LIN {X 0,Y 369.311,Z 529.296,A -85,B 0,C 180,E1 -12777.819,E2 -12777.819} C_VEL
LIN {X 0,Y 369.451,Z 529.279,A -85,B 0,C 180,E1 -12780,E2 -12780} C_VEL
LIN {X 0,Y 369.322,Z 529.581,A -85,B 0,C 180,E1 -12780.716,E2 -12780.716} C_VEL
LIN {X 0,Y 369.615,Z 530.776,A -85,B 0,C 180,E1 -12780.886,E2 -12780.886} C_VEL
LIN {X 0,Y 374.788,Z 542.535,A -85,B 0,C 180,E1 -12781.531,E2 -12781.531} C_VEL
LIN {X 0,Y 376.428,Z 547.392,A -85,B 0,C 180,E1 -12781.75,E2 -12781.75} C_VEL
LIN {X 0,Y 376.481,Z 569.423,A -85,B 0,C 180,E1 -12782.286,E2 -12782.286} C_VEL
LIN {X 0,Y 376.386,Z 581.867,A -85,B 0,C 180,E1 -12782.806,E2 -12782.806} C_VEL
LIN {X 0,Y 376.073,Z 593.193,A -85,B 0,C 180,E1 -12783.482,E2 -12783.482} C_VEL
LIN {X 0,Y 375.404,Z 605.188,A -85,B 0,C 180,E1 -12784.429,E2 -12784.429} C_VEL
LIN {X 0,Y 374.736,Z 615.62,A -85,B 0,C 180,E1 -12785.499,E2 -12785.499} C_VEL
LIN {X 0,Y 373.913,Z 625.309,A -85,B 0,C 180,E1 -12786.747,E2 -12786.747} C_VEL
LIN {X 0,Y 373.096,Z 633.924,A -85,B 0,C 180,E1 -12788.122,E2 -12788.122} C_VEL
LIN {X 0,Y 372.293,Z 640.997,A -85,B 0,C 180,E1 -12789.508,E2 -12789.508} C_VEL
LIN {X 0,Y 371.594,Z 646.791,A -85,B 0,C 180,E1 -12790.903,E2 -12790.903} C_VEL
LIN {X 0,Y 370.872,Z 652.348,A -85,B 0,C 180,E1 -12792.588,E2 -12792.588} C_VEL
LIN {X 0,Y 370.18,Z 657.037,A -85,B 0,C 180,E1 -12794.481,E2 -12794.481} C_VEL
LIN {X 0,Y 369.897,Z 658.839,A -85,B 0,C 180,E1 -12795.427,E2 -12795.427} C_VEL
LIN {X 0,Y 369.624,Z 660.529,A -85,B 0,C 180,E1 -12796.572,E2 -12796.572} C_VEL
LIN {X 0,Y 369.348,Z 661.936,A -85,B 0,C 180,E1 -12797.94,E2 -12797.94} C_VEL
LIN {X 0,Y 369.231,Z 662.502,A -85,B 0,C 180,E1 -12798.88,E2 -12798.88} C_VEL
LIN {X 0,Y 369.092,Z 662.755,A -85,B 0,C 180,E1 -12800.045,E2 -12800.045} C_VEL
LIN {X 0,Y 369.016,Z 662.563,A -85,B 0,C 180,E1 -12801.215,E2 -12801.215} C_VEL
LIN {X 0,Y 368.966,Z 661.866,A -85,B 0,C 180,E1 -12802.393,E2 -12802.393} C_VEL
LIN {X 0,Y 369.024,Z 660.255,A -85,B 0,C 180,E1 -12803.918,E2 -12803.918} C_VEL
LIN {X 0,Y 369.263,Z 656.737,A -85,B 0,C 180,E1 -12805.961,E2 -12805.961} C_VEL
LIN {X 0,Y 369.574,Z 652.281,A -85,B 0,C 180,E1 -12807.769,E2 -12807.769} C_VEL
LIN {X 0,Y 370.008,Z 646.26,A -85,B 0,C 180,E1 -12809.594,E2 -12809.594} C_VEL
LIN {X 0,Y 370.55,Z 638.583,A -85,B 0,C 180,E1 -12811.409,E2 -12811.409} C_VEL
LIN {X 0,Y 371.201,Z 630.13,A -85,B 0,C 180,E1 -12812.979,E2 -12812.979} C_VEL
LIN {X 0,Y 371.811,Z 620.701,A -85,B 0,C 180,E1 -12814.4,E2 -12814.4} C_VEL
LIN {X 0,Y 372.43,Z 610.239,A -85,B 0,C 180,E1 -12815.664,E2 -12815.664} C_VEL
LIN {X 0,Y 373.009,Z 599.015,A -85,B 0,C 180,E1 -12816.743,E2 -12816.743} C_VEL
LIN {X 0,Y 373.444,Z 588.322,A -85,B 0,C 180,E1 -12817.554,E2 -12817.554} C_VEL
LIN {X 0,Y 373.76,Z 575.886,A -85,B 0,C 180,E1 -12818.266,E2 -12818.266} C_VEL
LIN {X 0,Y 373.907,Z 562.29,A -85,B 0,C 180,E1 -12818.796,E2 -12818.796} C_VEL
LIN {X 0,Y 373.805,Z 544.593,A -85,B 0,C 180,E1 -12819.216,E2 -12819.216} C_VEL
LIN {X 0,Y 369.179,Z 530.472,A -85,B 0,C 180,E1 -12819.719,E2 -12819.719} C_VEL
LIN {X 0,Y 368.967,Z 529.473,A -85,B 0,C 180,E1 -12819.913,E2 -12819.913} C_VEL
LIN {X 0,Y 368.887,Z 529.349,A -85,B 0,C 180,E1 -12823.618,E2 -12823.618} C_VEL
LIN {X 0,Y 368.937,Z 529.338,A -85,B 0,C 180,E1 -12826.705,E2 -12826.705} C_VEL
LIN {X 0,Y 368.952,Z 529.339,A -85,B 0,C 180,E1 -12829.637,E2 -12829.637} C_VEL
LIN {X 0,Y 368.903,Z 529.345,A -85,B 0,C 180,E1 -12833.145,E2 -12833.145} C_VEL
LIN {X 0,Y 368.897,Z 529.342,A -85,B 0,C 180,E1 -12836.463,E2 -12836.463} C_VEL
LIN {X 0,Y 368.93,Z 529.34,A -85,B 0,C 180,E1 -12839.047,E2 -12839.047} C_VEL
LIN {X 0,Y 368.981,Z 529.338,A -85,B 0,C 180,E1 -12841.565,E2 -12841.565} C_VEL
LIN {X 0,Y 369.002,Z 529.331,A -85,B 0,C 180,E1 -12844.021,E2 -12844.021} C_VEL
LIN {X 0,Y 368.936,Z 529.344,A -85,B 0,C 180,E1 -12847.606,E2 -12847.606} C_VEL
LIN {X 0,Y 368.958,Z 529.336,A -85,B 0,C 180,E1 -12851.106,E2 -12851.106} C_VEL
LIN {X 0,Y 369.001,Z 529.329,A -85,B 0,C 180,E1 -12854.536,E2 -12854.536} C_VEL
LIN {X 0,Y 369.009,Z 529.332,A -85,B 0,C 180,E1 -12857.907,E2 -12857.907} C_VEL
LIN {X 0,Y 369.098,Z 529.319,A -85,B 0,C 180,E1 -12861.238,E2 -12861.238} C_VEL
LIN {X 0,Y 369.135,Z 529.313,A -85,B 0,C 180,E1 -12864.538,E2 -12864.538} C_VEL
LIN {X 0,Y 369.321,Z 529.295,A -85,B 0,C 180,E1 -12867.819,E2 -12867.819} C_VEL
LIN {X 0,Y 369.461,Z 529.276,A -85,B 0,C 180,E1 -12870,E2 -12870} C_VEL
LIN {X 0,Y 369.321,Z 529.292,A -85,B 0,C 180,E1 -12872.181,E2 -12872.181} C_VEL
LIN {X 0,Y 369.178,Z 529.308,A -85,B 0,C 180,E1 -12876.559,E2 -12876.559} C_VEL
LIN {X 0,Y 369.068,Z 529.327,A -85,B 0,C 180,E1 -12879.868,E2 -12879.868} C_VEL
LIN {X 0,Y 369.041,Z 529.33,A -85,B 0,C 180,E1 -12883.772,E2 -12883.772} C_VEL
LIN {X 0,Y 369.005,Z 529.334,A -85,B 0,C 180,E1 -12887.768,E2 -12887.768} C_VEL
LIN {X 0,Y 368.9,Z 529.341,A -85,B 0,C 180,E1 -12891.574,E2 -12891.574} C_VEL
LIN {X 0,Y 368.957,Z 529.335,A -85,B 0,C 180,E1 -12894.775,E2 -12894.775} C_VEL
LIN {X 0,Y 368.986,Z 529.334,A -85,B 0,C 180,E1 -12896.321,E2 -12896.321} C_VEL
LIN {X 0,Y 368.299,Z 529.418,A -85,B 0,C 180,E1 -12897.231,E2 -12897.231} C_VEL
LIN {X 0,Y 365.402,Z 529.778,A -85,B 0,C 180,E1 -12898.711,E2 -12898.711} C_VEL
LIN {X 0,Y 362.962,Z 530.087,A -85,B 0,C 180,E1 -12899.908,E2 -12899.908} C_VEL
LIN {X 0,Y 361.925,Z 530.211,A -85,B 0,C 180,E1 -12900.834,E2 -12900.834} C_VEL
LIN {X 0,Y 361.846,Z 530.221,A -85,B 0,C 180,E1 -12901.148,E2 -12901.148} C_VEL
LIN {X 0,Y 361.856,Z 530.223,A -85,B 0,C 180,E1 -12904.279,E2 -12904.279} C_VEL
LIN {X 0,Y 361.866,Z 530.218,A -85,B 0,C 180,E1 -12907.222,E2 -12907.222} C_VEL
LIN {X 0,Y 361.906,Z 530.214,A -85,B 0,C 180,E1 -12910.767,E2 -12910.767} C_VEL
LIN {X 0,Y 361.91,Z 530.216,A -85,B 0,C 180,E1 -12914.353,E2 -12914.353} C_VEL
LIN {X 0,Y 361.835,Z 530.223,A -85,B 0,C 180,E1 -12917.567,E2 -12917.567} C_VEL
LIN {X 0,Y 361.868,Z 530.218,A -85,B 0,C 180,E1 -12920.972,E2 -12920.972} C_VEL
LIN {X 0,Y 361.871,Z 530.219,A -85,B 0,C 180,E1 -12924.654,E2 -12924.654} C_VEL
LIN {X 0,Y 361.857,Z 530.224,A -85,B 0,C 180,E1 -12928.372,E2 -12928.372} C_VEL
LIN {X 0,Y 361.919,Z 530.218,A -85,B 0,C 180,E1 -12932.221,E2 -12932.221} C_VEL
LIN {X 0,Y 361.923,Z 530.213,A -85,B 0,C 180,E1 -12934.709,E2 -12934.709} C_VEL
LIN {X 0,Y 361.894,Z 530.221,A -85,B 0,C 180,E1 -12938.347,E2 -12938.347} C_VEL
LIN {X 0,Y 361.962,Z 530.21,A -85,B 0,C 180,E1 -12942.06,E2 -12942.06} C_VEL
LIN {X 0,Y 361.992,Z 530.206,A -85,B 0,C 180,E1 -12946.1,E2 -12946.1} C_VEL
LIN {X 0,Y 362.029,Z 530.2,A -85,B 0,C 180,E1 -12949.937,E2 -12949.937} C_VEL
LIN {X 0,Y 362.145,Z 530.187,A -85,B 0,C 180,E1 -12952.192,E2 -12952.192} C_VEL
LIN {X 0,Y 362.113,Z 530.194,A -85,B 0,C 180,E1 -12954.431,E2 -12954.431} C_VEL
LIN {X 0,Y 362.276,Z 530.168,A -85,B 0,C 180,E1 -12957.776,E2 -12957.776} C_VEL
LIN {X 0,Y 362.42,Z 530.151,A -85,B 0,C 180,E1 -12960,E2 -12960} C_VEL
LIN {X 0,Y 362.275,Z 530.171,A -85,B 0,C 180,E1 -12962.223,E2 -12962.223} C_VEL
LIN {X 0,Y 362.155,Z 530.187,A -85,B 0,C 180,E1 -12966.686,E2 -12966.686} C_VEL
LIN {X 0,Y 362.023,Z 530.2,A -85,B 0,C 180,E1 -12970.062,E2 -12970.062} C_VEL
LIN {X 0,Y 361.99,Z 530.203,A -85,B 0,C 180,E1 -12973.899,E2 -12973.899} C_VEL
LIN {X 0,Y 361.96,Z 530.207,A -85,B 0,C 180,E1 -12977.939,E2 -12977.939} C_VEL
LIN {X 0,Y 361.854,Z 530.219,A -85,B 0,C 180,E1 -12981.655,E2 -12981.655} C_VEL
LIN {X 0,Y 361.92,Z 530.212,A -85,B 0,C 180,E1 -12985.29,E2 -12985.29} C_VEL
LIN {X 0,Y 361.916,Z 530.212,A -85,B 0,C 180,E1 -12987.778,E2 -12987.778} C_VEL
LIN {X 0,Y 361.84,Z 530.223,A -85,B 0,C 180,E1 -12991.285,E2 -12991.285} C_VEL
LIN {X 0,Y 361.848,Z 530.222,A -85,B 0,C 180,E1 -12994.281,E2 -12994.281} C_VEL
LIN {X 0,Y 361.859,Z 530.221,A -85,B 0,C 180,E1 -12997.223,E2 -12997.223} C_VEL
LIN {X 0,Y 361.83,Z 530.228,A -85,B 0,C 180,E1 -13000.756,E2 -13000.756} C_VEL
LIN {X 0,Y 361.83,Z 530.224,A -85,B 0,C 180,E1 -13004.366,E2 -13004.366} C_VEL
LIN {X 0,Y 361.832,Z 530.223,A -85,B 0,C 180,E1 -13007.568,E2 -13007.568} C_VEL
LIN {X 0,Y 361.868,Z 530.224,A -85,B 0,C 180,E1 -13010.973,E2 -13010.973} C_VEL
LIN {X 0,Y 361.875,Z 530.224,A -85,B 0,C 180,E1 -13014.655,E2 -13014.655} C_VEL
LIN {X 0,Y 361.97,Z 530.418,A -85,B 0,C 180,E1 -13015.791,E2 -13015.791} C_VEL
LIN {X 0,Y 364.841,Z 544.913,A -85,B 0,C 180,E1 -13019.626,E2 -13019.626} C_VEL
LIN {X 0,Y 365.525,Z 550.193,A -85,B 0,C 180,E1 -13020.956,E2 -13020.956} C_VEL
LIN {X 0,Y 364.093,Z 565.356,A -85,B 0,C 180,E1 -13024.566,E2 -13024.566} C_VEL
LIN {X 0,Y 362.582,Z 584.16,A -85,B 0,C 180,E1 -13028.987,E2 -13028.987} C_VEL
LIN {X 0,Y 361.692,Z 599.262,A -85,B 0,C 180,E1 -13032.463,E2 -13032.463} C_VEL
LIN {X 0,Y 363.071,Z 616.076,A -85,B 0,C 180,E1 -13032.992,E2 -13032.992} C_VEL
LIN {X 0,Y 365.581,Z 647.576,A -85,B 0,C 180,E1 -13033.892,E2 -13033.892} C_VEL
LIN {X 0,Y 364.865,Z 683.205,A -85,B 0,C 180,E1 -13034.821,E2 -13034.821} C_VEL
LIN {X 0,Y 364.369,Z 695.019,A -85,B 0,C 180,E1 -13035.336,E2 -13035.336} C_VEL
LIN {X 0,Y 363.573,Z 705.872,A -85,B 0,C 180,E1 -13036.018,E2 -13036.018} C_VEL
LIN {X 0,Y 363.02,Z 715.883,A -85,B 0,C 180,E1 -13036.852,E2 -13036.852} C_VEL
LIN {X 0,Y 362.191,Z 726.2,A -85,B 0,C 180,E1 -13037.96,E2 -13037.96} C_VEL
LIN {X 0,Y 361.582,Z 734.455,A -85,B 0,C 180,E1 -13039.076,E2 -13039.076} C_VEL
LIN {X 0,Y 361.212,Z 742.776,A -85,B 0,C 180,E1 -13040.481,E2 -13040.481} C_VEL
LIN {X 0,Y 361.042,Z 749.412,A -85,B 0,C 180,E1 -13041.887,E2 -13041.887} C_VEL
LIN {X 0,Y 361.026,Z 754.682,A -85,B 0,C 180,E1 -13043.293,E2 -13043.293} C_VEL
LIN {X 0,Y 361.121,Z 759.526,A -85,B 0,C 180,E1 -13044.976,E2 -13044.976} C_VEL
LIN {X 0,Y 361.292,Z 762.876,A -85,B 0,C 180,E1 -13046.654,E2 -13046.654} C_VEL
LIN {X 0,Y 361.355,Z 764.387,A -85,B 0,C 180,E1 -13047.771,E2 -13047.771} C_VEL
LIN {X 0,Y 361.435,Z 765.3,A -85,B 0,C 180,E1 -13048.886,E2 -13048.886} C_VEL
LIN {X 0,Y 361.683,Z 765.721,A -85,B 0,C 180,E1 -13050,E2 -13050} C_VEL
LIN {X 0,Y 361.405,Z 765.487,A -85,B 0,C 180,E1 -13051.114,E2 -13051.114} C_VEL
LIN {X 0,Y 361.299,Z 764.759,A -85,B 0,C 180,E1 -13052.229,E2 -13052.229} C_VEL
LIN {X 0,Y 361.247,Z 763.478,A -85,B 0,C 180,E1 -13053.346,E2 -13053.346} C_VEL
LIN {X 0,Y 361.011,Z 760.507,A -85,B 0,C 180,E1 -13055.026,E2 -13055.026} C_VEL
LIN {X 0,Y 360.857,Z 756.183,A -85,B 0,C 180,E1 -13056.71,E2 -13056.71} C_VEL
LIN {X 0,Y 360.96,Z 750.431,A -85,B 0,C 180,E1 -13058.396,E2 -13058.396} C_VEL
LIN {X 0,Y 361.297,Z 742.939,A -85,B 0,C 180,E1 -13060.082,E2 -13060.082} C_VEL
LIN {X 0,Y 361.872,Z 735.075,A -85,B 0,C 180,E1 -13061.482,E2 -13061.482} C_VEL
LIN {X 0,Y 362.806,Z 725.285,A -85,B 0,C 180,E1 -13062.871,E2 -13062.871} C_VEL
LIN {X 0,Y 363.901,Z 714.064,A -85,B 0,C 180,E1 -13064.112,E2 -13064.112} C_VEL
LIN {X 0,Y 364.995,Z 702.831,A -85,B 0,C 180,E1 -13065.066,E2 -13065.066} C_VEL
LIN {X 0,Y 365.976,Z 690.812,A -85,B 0,C 180,E1 -13065.832,E2 -13065.832} C_VEL
LIN {X 0,Y 366.787,Z 678.323,A -85,B 0,C 180,E1 -13066.387,E2 -13066.387} C_VEL
LIN {X 0,Y 367.347,Z 657.774,A -85,B 0,C 180,E1 -13066.933,E2 -13066.933} C_VEL
LIN {X 0,Y 367.41,Z 645.582,A -85,B 0,C 180,E1 -13067.245,E2 -13067.245} C_VEL
LIN {X 0,Y 365.873,Z 619.079,A -85,B 0,C 180,E1 -13068.042,E2 -13068.042} C_VEL
LIN {X 0,Y 363.361,Z 597.729,A -85,B 0,C 180,E1 -13068.795,E2 -13068.795} C_VEL
LIN {X 0,Y 361.865,Z 587.816,A -85,B 0,C 180,E1 -13069.216,E2 -13069.216} C_VEL
LIN {X 0,Y 362.492,Z 575.864,A -85,B 0,C 180,E1 -13071.914,E2 -13071.914} C_VEL
LIN {X 0,Y 363.779,Z 558.36,A -85,B 0,C 180,E1 -13076.072,E2 -13076.072} C_VEL
LIN {X 0,Y 364.81,Z 547.337,A -85,B 0,C 180,E1 -13078.79,E2 -13078.79} C_VEL
LIN {X 0,Y 364.315,Z 542.419,A -85,B 0,C 180,E1 -13080.103,E2 -13080.103} C_VEL
LIN {X 0,Y 362.061,Z 530.888,A -85,B 0,C 180,E1 -13083.418,E2 -13083.418} C_VEL
LIN {X 0,Y 361.927,Z 530.221,A -85,B 0,C 180,E1 -13083.776,E2 -13083.776} C_VEL
LIN {X 0,Y 361.86,Z 530.224,A -85,B 0,C 180,E1 -13087.223,E2 -13087.223} C_VEL
LIN {X 0,Y 361.831,Z 530.226,A -85,B 0,C 180,E1 -13090.755,E2 -13090.755} C_VEL
LIN {X 0,Y 361.842,Z 530.223,A -85,B 0,C 180,E1 -13094.363,E2 -13094.363} C_VEL
LIN {X 0,Y 361.878,Z 530.214,A -85,B 0,C 180,E1 -13097.559,E2 -13097.559} C_VEL
LIN {X 0,Y 361.87,Z 530.217,A -85,B 0,C 180,E1 -13100.971,E2 -13100.971} C_VEL
LIN {X 0,Y 361.868,Z 530.216,A -85,B 0,C 180,E1 -13104.655,E2 -13104.655} C_VEL
LIN {X 0,Y 361.853,Z 530.22,A -85,B 0,C 180,E1 -13108.372,E2 -13108.372} C_VEL
LIN {X 0,Y 361.915,Z 530.215,A -85,B 0,C 180,E1 -13112.222,E2 -13112.222} C_VEL
LIN {X 0,Y 361.92,Z 530.213,A -85,B 0,C 180,E1 -13114.71,E2 -13114.71} C_VEL
LIN {X 0,Y 361.885,Z 530.22,A -85,B 0,C 180,E1 -13118.347,E2 -13118.347} C_VEL
LIN {X 0,Y 361.959,Z 530.207,A -85,B 0,C 180,E1 -13122.061,E2 -13122.061} C_VEL
LIN {X 0,Y 361.99,Z 530.207,A -85,B 0,C 180,E1 -13126.101,E2 -13126.101} C_VEL
LIN {X 0,Y 362.028,Z 530.203,A -85,B 0,C 180,E1 -13129.938,E2 -13129.938} C_VEL
LIN {X 0,Y 362.143,Z 530.19,A -85,B 0,C 180,E1 -13132.193,E2 -13132.193} C_VEL
LIN {X 0,Y 362.116,Z 530.191,A -85,B 0,C 180,E1 -13134.432,E2 -13134.432} C_VEL
LIN {X 0,Y 362.275,Z 530.173,A -85,B 0,C 180,E1 -13137.777,E2 -13137.777} C_VEL
LIN {X 0,Y 362.391,Z 530.263,A -85,B 0,C 180,E1 -13140.125,E2 -13140.125} C_VEL
LIN {X 0,Y 362.532,Z 531.164,A -85,B 0,C 180,E1 -13140.344,E2 -13140.344} C_VEL
LIN {X 0,Y 368.491,Z 544.802,A -85,B 0,C 180,E1 -13141.139,E2 -13141.139} C_VEL
LIN {X 0,Y 369.944,Z 548.817,A -85,B 0,C 180,E1 -13141.334,E2 -13141.334} C_VEL
LIN {X 0,Y 370.011,Z 570.604,A -85,B 0,C 180,E1 -13141.875,E2 -13141.875} C_VEL
LIN {X 0,Y 369.898,Z 583.228,A -85,B 0,C 180,E1 -13142.413,E2 -13142.413} C_VEL
LIN {X 0,Y 369.509,Z 595.258,A -85,B 0,C 180,E1 -13143.157,E2 -13143.157} C_VEL
LIN {X 0,Y 368.803,Z 606.791,A -85,B 0,C 180,E1 -13144.098,E2 -13144.098} C_VEL
LIN {X 0,Y 368.09,Z 617.219,A -85,B 0,C 180,E1 -13145.204,E2 -13145.204} C_VEL
LIN {X 0,Y 367.12,Z 627.66,A -85,B 0,C 180,E1 -13146.596,E2 -13146.596} C_VEL
LIN {X 0,Y 366.269,Z 636.06,A -85,B 0,C 180,E1 -13147.997,E2 -13147.997} C_VEL
LIN {X 0,Y 365.246,Z 644.156,A -85,B 0,C 180,E1 -13149.693,E2 -13149.693} C_VEL
LIN {X 0,Y 364.561,Z 649.571,A -85,B 0,C 180,E1 -13151.115,E2 -13151.115} C_VEL
LIN {X 0,Y 363.801,Z 654.789,A -85,B 0,C 180,E1 -13152.836,E2 -13152.836} C_VEL
LIN {X 0,Y 363.165,Z 658.84,A -85,B 0,C 180,E1 -13154.629,E2 -13154.629} C_VEL
LIN {X 0,Y 362.845,Z 660.682,A -85,B 0,C 180,E1 -13155.734,E2 -13155.734} C_VEL
LIN {X 0,Y 362.552,Z 662.185,A -85,B 0,C 180,E1 -13156.905,E2 -13156.905} C_VEL
LIN {X 0,Y 362.314,Z 663.202,A -85,B 0,C 180,E1 -13158.111,E2 -13158.111} C_VEL
LIN {X 0,Y 362.171,Z 663.712,A -85,B 0,C 180,E1 -13159.262,E2 -13159.262} C_VEL
LIN {X 0,Y 361.999,Z 663.563,A -85,B 0,C 180,E1 -13161.272,E2 -13161.272} C_VEL
LIN {X 0,Y 361.945,Z 662.47,A -85,B 0,C 180,E1 -13162.852,E2 -13162.852} C_VEL
LIN {X 0,Y 362.032,Z 660.894,A -85,B 0,C 180,E1 -13164.165,E2 -13164.165} C_VEL
LIN {X 0,Y 362.221,Z 657.929,A -85,B 0,C 180,E1 -13165.885,E2 -13165.885} C_VEL
LIN {X 0,Y 362.542,Z 653.515,A -85,B 0,C 180,E1 -13167.727,E2 -13167.727} C_VEL
LIN {X 0,Y 363.012,Z 647.024,A -85,B 0,C 180,E1 -13169.731,E2 -13169.731} C_VEL
LIN {X 0,Y 363.555,Z 639.803,A -85,B 0,C 180,E1 -13171.463,E2 -13171.463} C_VEL
LIN {X 0,Y 364.19,Z 631.558,A -85,B 0,C 180,E1 -13173.036,E2 -13173.036} C_VEL
LIN {X 0,Y 364.843,Z 621.635,A -85,B 0,C 180,E1 -13174.563,E2 -13174.563} C_VEL
LIN {X 0,Y 365.488,Z 611.245,A -85,B 0,C 180,E1 -13175.838,E2 -13175.838} C_VEL
LIN {X 0,Y 366.053,Z 600.766,A -85,B 0,C 180,E1 -13176.869,E2 -13176.869} C_VEL
LIN {X 0,Y 366.543,Z 589.314,A -85,B 0,C 180,E1 -13177.761,E2 -13177.761} C_VEL
LIN {X 0,Y 366.86,Z 577.017,A -85,B 0,C 180,E1 -13178.478,E2 -13178.478} C_VEL
LIN {X 0,Y 367.009,Z 563.458,A -85,B 0,C 180,E1 -13179.02,E2 -13179.02} C_VEL
LIN {X 0,Y 366.849,Z 545.757,A -85,B 0,C 180,E1 -13179.453,E2 -13179.453} C_VEL
LIN {X 0,Y 362.055,Z 531.081,A -85,B 0,C 180,E1 -13180.003,E2 -13180.003} C_VEL
LIN {X 0,Y 361.897,Z 530.288,A -85,B 0,C 180,E1 -13180.221,E2 -13180.221} C_VEL
LIN {X 0,Y 361.836,Z 530.225,A -85,B 0,C 180,E1 -13184.058,E2 -13184.058} C_VEL
LIN {X 0,Y 361.88,Z 530.221,A -85,B 0,C 180,E1 -13187.179,E2 -13187.179} C_VEL
LIN {X 0,Y 361.88,Z 530.217,A -85,B 0,C 180,E1 -13190.143,E2 -13190.143} C_VEL
LIN {X 0,Y 361.869,Z 530.22,A -85,B 0,C 180,E1 -13192.983,E2 -13192.983} C_VEL
LIN {X 0,Y 361.859,Z 530.219,A -85,B 0,C 180,E1 -13196.632,E2 -13196.632} C_VEL
LIN {X 0,Y 361.876,Z 530.221,A -85,B 0,C 180,E1 -13199.673,E2 -13199.673} C_VEL
LIN {X 0,Y 361.957,Z 530.213,A -85,B 0,C 180,E1 -13203.476,E2 -13203.476} C_VEL
LIN {X 0,Y 361.893,Z 530.217,A -85,B 0,C 180,E1 -13207.146,E2 -13207.146} C_VEL
LIN {X 0,Y 361.89,Z 530.215,A -85,B 0,C 180,E1 -13210.723,E2 -13210.723} C_VEL
LIN {X 0,Y 361.947,Z 530.209,A -85,B 0,C 180,E1 -13214.227,E2 -13214.227} C_VEL
LIN {X 0,Y 362.003,Z 530.201,A -85,B 0,C 180,E1 -13216.528,E2 -13216.528} C_VEL
LIN {X 0,Y 362.035,Z 530.201,A -85,B 0,C 180,E1 -13219.938,E2 -13219.938} C_VEL
LIN {X 0,Y 362.14,Z 530.187,A -85,B 0,C 180,E1 -13223.313,E2 -13223.313} C_VEL
LIN {X 0,Y 362.285,Z 530.172,A -85,B 0,C 180,E1 -13227.777,E2 -13227.777} C_VEL
LIN {X 0,Y 362.431,Z 530.151,A -85,B 0,C 180,E1 -13230,E2 -13230} C_VEL
LIN {X 0,Y 362.285,Z 530.168,A -85,B 0,C 180,E1 -13232.224,E2 -13232.224} C_VEL
LIN {X 0,Y 362.14,Z 530.184,A -85,B 0,C 180,E1 -13236.687,E2 -13236.687} C_VEL
LIN {X 0,Y 362.005,Z 530.205,A -85,B 0,C 180,E1 -13240.063,E2 -13240.063} C_VEL
LIN {X 0,Y 362.002,Z 530.207,A -85,B 0,C 180,E1 -13243.898,E2 -13243.898} C_VEL
LIN {X 0,Y 361.971,Z 530.211,A -85,B 0,C 180,E1 -13247.938,E2 -13247.938} C_VEL
LIN {X 0,Y 361.864,Z 530.222,A -85,B 0,C 180,E1 -13251.654,E2 -13251.654} C_VEL
LIN {X 0,Y 361.929,Z 530.211,A -85,B 0,C 180,E1 -13255.289,E2 -13255.289} C_VEL
LIN {X 0,Y 361.91,Z 530.217,A -85,B 0,C 180,E1 -13257.778,E2 -13257.778} C_VEL
LIN {X 0,Y 361.846,Z 530.221,A -85,B 0,C 180,E1 -13261.148,E2 -13261.148} C_VEL
LIN {X 0,Y 361.196,Z 530.307,A -85,B 0,C 180,E1 -13262.076,E2 -13262.076} C_VEL
LIN {X 0,Y 358.359,Z 530.659,A -85,B 0,C 180,E1 -13263.586,E2 -13263.586} C_VEL
LIN {X 0,Y 355.942,Z 530.959,A -85,B 0,C 180,E1 -13264.807,E2 -13264.807} C_VEL
LIN {X 0,Y 354.894,Z 531.09,A -85,B 0,C 180,E1 -13265.752,E2 -13265.752} C_VEL
LIN {X 0,Y 354.804,Z 531.099,A -85,B 0,C 180,E1 -13266.072,E2 -13266.072} C_VEL
LIN {X 0,Y 354.824,Z 531.096,A -85,B 0,C 180,E1 -13269.423,E2 -13269.423} C_VEL
LIN {X 0,Y 354.837,Z 531.094,A -85,B 0,C 180,E1 -13272.875,E2 -13272.875} C_VEL
LIN {X 0,Y 354.783,Z 531.107,A -85,B 0,C 180,E1 -13276.105,E2 -13276.105} C_VEL
LIN {X 0,Y 354.786,Z 531.1,A -85,B 0,C 180,E1 -13279.178,E2 -13279.178} C_VEL
LIN {X 0,Y 354.805,Z 531.102,A -85,B 0,C 180,E1 -13282.401,E2 -13282.401} C_VEL
LIN {X 0,Y 354.809,Z 531.098,A -85,B 0,C 180,E1 -13284.94,E2 -13284.94} C_VEL
LIN {X 0,Y 354.813,Z 531.101,A -85,B 0,C 180,E1 -13288.398,E2 -13288.398} C_VEL
LIN {X 0,Y 354.851,Z 531.093,A -85,B 0,C 180,E1 -13291.619,E2 -13291.619} C_VEL
LIN {X 0,Y 354.895,Z 531.092,A -85,B 0,C 180,E1 -13294.172,E2 -13294.172} C_VEL
LIN {X 0,Y 354.834,Z 531.096,A -85,B 0,C 180,E1 -13297.893,E2 -13297.893} C_VEL
LIN {X 0,Y 354.918,Z 531.086,A -85,B 0,C 180,E1 -13301.89,E2 -13301.89} C_VEL
LIN {X 0,Y 354.937,Z 531.084,A -85,B 0,C 180,E1 -13305.98,E2 -13305.98} C_VEL
LIN {X 0,Y 354.976,Z 531.077,A -85,B 0,C 180,E1 -13309.735,E2 -13309.735} C_VEL
LIN {X 0,Y 355.108,Z 531.063,A -85,B 0,C 180,E1 -13312.036,E2 -13312.036} C_VEL
LIN {X 0,Y 355.087,Z 531.068,A -85,B 0,C 180,E1 -13314.32,E2 -13314.32} C_VEL
LIN {X 0,Y 355.239,Z 531.044,A -85,B 0,C 180,E1 -13317.732,E2 -13317.732} C_VEL
LIN {X 0,Y 355.39,Z 531.027,A -85,B 0,C 180,E1 -13320,E2 -13320} C_VEL
LIN {X 0,Y 355.238,Z 531.048,A -85,B 0,C 180,E1 -13322.267,E2 -13322.267} C_VEL
LIN {X 0,Y 355.119,Z 531.062,A -85,B 0,C 180,E1 -13326.819,E2 -13326.819} C_VEL
LIN {X 0,Y 354.97,Z 531.08,A -85,B 0,C 180,E1 -13330.264,E2 -13330.264} C_VEL
LIN {X 0,Y 354.935,Z 531.083,A -85,B 0,C 180,E1 -13334.018,E2 -13334.018} C_VEL
LIN {X 0,Y 354.916,Z 531.085,A -85,B 0,C 180,E1 -13338.109,E2 -13338.109} C_VEL
LIN {X 0,Y 354.81,Z 531.098,A -85,B 0,C 180,E1 -13342.107,E2 -13342.107} C_VEL
LIN {X 0,Y 354.892,Z 531.087,A -85,B 0,C 180,E1 -13345.828,E2 -13345.828} C_VEL
LIN {X 0,Y 354.848,Z 531.092,A -85,B 0,C 180,E1 -13349.679,E2 -13349.679} C_VEL
LIN {X 0,Y 354.8,Z 531.098,A -85,B 0,C 180,E1 -13353.702,E2 -13353.702} C_VEL
LIN {X 0,Y 354.793,Z 531.102,A -85,B 0,C 180,E1 -13356.46,E2 -13356.46} C_VEL
LIN {X 0,Y 354.819,Z 531.097,A -85,B 0,C 180,E1 -13359.424,E2 -13359.424} C_VEL
LIN {X 0,Y 354.783,Z 531.107,A -85,B 0,C 180,E1 -13362.868,E2 -13362.868} C_VEL
LIN {X 0,Y 354.772,Z 531.102,A -85,B 0,C 180,E1 -13366.106,E2 -13366.106} C_VEL
LIN {X 0,Y 354.785,Z 531.104,A -85,B 0,C 180,E1 -13369.18,E2 -13369.18} C_VEL
LIN {X 0,Y 354.805,Z 531.099,A -85,B 0,C 180,E1 -13372.403,E2 -13372.403} C_VEL
LIN {X 0,Y 354.897,Z 531.194,A -85,B 0,C 180,E1 -13375.534,E2 -13375.534} C_VEL
LIN {X 0,Y 357.57,Z 544.872,A -85,B 0,C 180,E1 -13379.268,E2 -13379.268} C_VEL
LIN {X 0,Y 358.49,Z 550.201,A -85,B 0,C 180,E1 -13380.653,E2 -13380.653} C_VEL
LIN {X 0,Y 357.406,Z 561.546,A -85,B 0,C 180,E1 -13383.427,E2 -13383.427} C_VEL
LIN {X 0,Y 356.159,Z 575.321,A -85,B 0,C 180,E1 -13386.756,E2 -13386.756} C_VEL
LIN {X 0,Y 355.091,Z 590.262,A -85,B 0,C 180,E1 -13390.339,E2 -13390.339} C_VEL
LIN {X 0,Y 354.643,Z 598.077,A -85,B 0,C 180,E1 -13392.154,E2 -13392.154} C_VEL
LIN {X 0,Y 355.236,Z 605.679,A -85,B 0,C 180,E1 -13392.427,E2 -13392.427} C_VEL
LIN {X 0,Y 358.62,Z 648.08,A -85,B 0,C 180,E1 -13393.675,E2 -13393.675} C_VEL
LIN {X 0,Y 357.919,Z 682.222,A -85,B 0,C 180,E1 -13394.592,E2 -13394.592} C_VEL
LIN {X 0,Y 357.424,Z 693.991,A -85,B 0,C 180,E1 -13395.117,E2 -13395.117} C_VEL
LIN {X 0,Y 356.534,Z 705.776,A -85,B 0,C 180,E1 -13395.881,E2 -13395.881} C_VEL
LIN {X 0,Y 355.835,Z 716.938,A -85,B 0,C 180,E1 -13396.872,E2 -13396.872} C_VEL
LIN {X 0,Y 355.132,Z 725.731,A -85,B 0,C 180,E1 -13397.862,E2 -13397.862} C_VEL
LIN {X 0,Y 354.475,Z 734.768,A -85,B 0,C 180,E1 -13399.144,E2 -13399.144} C_VEL
LIN {X 0,Y 354.109,Z 742.833,A -85,B 0,C 180,E1 -13400.576,E2 -13400.576} C_VEL
LIN {X 0,Y 353.951,Z 750.49,A -85,B 0,C 180,E1 -13402.326,E2 -13402.326} C_VEL
LIN {X 0,Y 353.981,Z 755.676,A -85,B 0,C 180,E1 -13403.884,E2 -13403.884} C_VEL
LIN {X 0,Y 354.136,Z 759.618,A -85,B 0,C 180,E1 -13405.447,E2 -13405.447} C_VEL
LIN {X 0,Y 354.249,Z 761.746,A -85,B 0,C 180,E1 -13406.588,E2 -13406.588} C_VEL
LIN {X 0,Y 354.319,Z 763.286,A -85,B 0,C 180,E1 -13407.726,E2 -13407.726} C_VEL
LIN {X 0,Y 354.405,Z 764.232,A -85,B 0,C 180,E1 -13408.864,E2 -13408.864} C_VEL
LIN {X 0,Y 354.654,Z 764.685,A -85,B 0,C 180,E1 -13410,E2 -13410} C_VEL
LIN {X 0,Y 354.368,Z 764.472,A -85,B 0,C 180,E1 -13411.136,E2 -13411.136} C_VEL
LIN {X 0,Y 354.25,Z 763.78,A -85,B 0,C 180,E1 -13412.274,E2 -13412.274} C_VEL
LIN {X 0,Y 354.198,Z 762.522,A -85,B 0,C 180,E1 -13413.412,E2 -13413.412} C_VEL
LIN {X 0,Y 353.926,Z 759.6,A -85,B 0,C 180,E1 -13415.126,E2 -13415.126} C_VEL
LIN {X 0,Y 353.772,Z 755.327,A -85,B 0,C 180,E1 -13416.845,E2 -13416.845} C_VEL
LIN {X 0,Y 353.918,Z 749.635,A -85,B 0,C 180,E1 -13418.565,E2 -13418.565} C_VEL
LIN {X 0,Y 354.169,Z 743.58,A -85,B 0,C 180,E1 -13419.999,E2 -13419.999} C_VEL
LIN {X 0,Y 354.686,Z 736.13,A -85,B 0,C 180,E1 -13421.428,E2 -13421.428} C_VEL
LIN {X 0,Y 355.658,Z 726.949,A -85,B 0,C 180,E1 -13422.844,E2 -13422.844} C_VEL
LIN {X 0,Y 356.772,Z 716.584,A -85,B 0,C 180,E1 -13424.109,E2 -13424.109} C_VEL
LIN {X 0,Y 357.806,Z 706.381,A -85,B 0,C 180,E1 -13425.085,E2 -13425.085} C_VEL
LIN {X 0,Y 358.913,Z 695.234,A -85,B 0,C 180,E1 -13425.91,E2 -13425.91} C_VEL
LIN {X 0,Y 359.936,Z 682.463,A -85,B 0,C 180,E1 -13426.594,E2 -13426.594} C_VEL
LIN {X 0,Y 360.389,Z 671.024,A -85,B 0,C 180,E1 -13427.008,E2 -13427.008} C_VEL
LIN {X 0,Y 360.868,Z 646.951,A -85,B 0,C 180,E1 -13427.624,E2 -13427.624} C_VEL
LIN {X 0,Y 359.336,Z 619.952,A -85,B 0,C 180,E1 -13428.468,E2 -13428.468} C_VEL
LIN {X 0,Y 357.013,Z 599.442,A -85,B 0,C 180,E1 -13429.215,E2 -13429.215} C_VEL
LIN {X 0,Y 354.904,Z 586.246,A -85,B 0,C 180,E1 -13429.785,E2 -13429.785} C_VEL
LIN {X 0,Y 354.968,Z 583.756,A -85,B 0,C 180,E1 -13430.272,E2 -13430.272} C_VEL
LIN {X 0,Y 355.962,Z 568.68,A -85,B 0,C 180,E1 -13433.874,E2 -13433.874} C_VEL
LIN {X 0,Y 357.376,Z 553.009,A -85,B 0,C 180,E1 -13437.755,E2 -13437.755} C_VEL
LIN {X 0,Y 357.857,Z 547.848,A -85,B 0,C 180,E1 -13439.082,E2 -13439.082} C_VEL
LIN {X 0,Y 356.752,Z 540.477,A -85,B 0,C 180,E1 -13441.139,E2 -13441.139} C_VEL
LIN {X 0,Y 354.909,Z 531.308,A -85,B 0,C 180,E1 -13443.92,E2 -13443.92} C_VEL
LIN {X 0,Y 354.804,Z 531.103,A -85,B 0,C 180,E1 -13447.597,E2 -13447.597} C_VEL
LIN {X 0,Y 354.783,Z 531.106,A -85,B 0,C 180,E1 -13451.171,E2 -13451.171} C_VEL
LIN {X 0,Y 354.811,Z 531.098,A -85,B 0,C 180,E1 -13454.514,E2 -13454.514} C_VEL
LIN {X 0,Y 354.832,Z 531.091,A -85,B 0,C 180,E1 -13457.669,E2 -13457.669} C_VEL
LIN {X 0,Y 354.847,Z 531.092,A -85,B 0,C 180,E1 -13460.671,E2 -13460.671} C_VEL
LIN {X 0,Y 354.816,Z 531.093,A -85,B 0,C 180,E1 -13464.3,E2 -13464.3} C_VEL
LIN {X 0,Y 354.791,Z 531.097,A -85,B 0,C 180,E1 -13467.667,E2 -13467.667} C_VEL
LIN {X 0,Y 354.862,Z 531.089,A -85,B 0,C 180,E1 -13470.621,E2 -13470.621} C_VEL
LIN {X 0,Y 354.891,Z 531.084,A -85,B 0,C 180,E1 -13474.172,E2 -13474.172} C_VEL
LIN {X 0,Y 354.828,Z 531.098,A -85,B 0,C 180,E1 -13477.894,E2 -13477.894} C_VEL
LIN {X 0,Y 354.914,Z 531.085,A -85,B 0,C 180,E1 -13481.892,E2 -13481.892} C_VEL
LIN {X 0,Y 354.935,Z 531.085,A -85,B 0,C 180,E1 -13485.981,E2 -13485.981} C_VEL
LIN {X 0,Y 354.975,Z 531.082,A -85,B 0,C 180,E1 -13489.736,E2 -13489.736} C_VEL
LIN {X 0,Y 355.106,Z 531.066,A -85,B 0,C 180,E1 -13492.037,E2 -13492.037} C_VEL
LIN {X 0,Y 355.09,Z 531.067,A -85,B 0,C 180,E1 -13494.321,E2 -13494.321} C_VEL
LIN {X 0,Y 355.239,Z 531.05,A -85,B 0,C 180,E1 -13497.733,E2 -13497.733} C_VEL
LIN {X 0,Y 355.306,Z 531.174,A -85,B 0,C 180,E1 -13499.575,E2 -13499.575} C_VEL
LIN {X 0,Y 355.521,Z 532.052,A -85,B 0,C 180,E1 -13499.788,E2 -13499.788} C_VEL
LIN {X 0,Y 361.746,Z 545.801,A -85,B 0,C 180,E1 -13500.654,E2 -13500.654} C_VEL
LIN {X 0,Y 363.471,Z 550.476,A -85,B 0,C 180,E1 -13500.899,E2 -13500.899} C_VEL
LIN {X 0,Y 363.547,Z 573.034,A -85,B 0,C 180,E1 -13501.492,E2 -13501.492} C_VEL
LIN {X 0,Y 363.428,Z 585.328,A -85,B 0,C 180,E1 -13502.047,E2 -13502.047} C_VEL
LIN {X 0,Y 363.004,Z 596.748,A -85,B 0,C 180,E1 -13502.775,E2 -13502.775} C_VEL
LIN {X 0,Y 362.248,Z 608.477,A -85,B 0,C 180,E1 -13503.755,E2 -13503.755} C_VEL
LIN {X 0,Y 361.471,Z 618.804,A -85,B 0,C 180,E1 -13504.88,E2 -13504.88} C_VEL
LIN {X 0,Y 360.522,Z 628.459,A -85,B 0,C 180,E1 -13506.192,E2 -13506.192} C_VEL
LIN {X 0,Y 359.624,Z 636.709,A -85,B 0,C 180,E1 -13507.581,E2 -13507.581} C_VEL
LIN {X 0,Y 358.54,Z 644.877,A -85,B 0,C 180,E1 -13509.307,E2 -13509.307} C_VEL
LIN {X 0,Y 357.748,Z 650.574,A -85,B 0,C 180,E1 -13510.817,E2 -13510.817} C_VEL
LIN {X 0,Y 356.997,Z 655.636,A -85,B 0,C 180,E1 -13512.507,E2 -13512.507} C_VEL
LIN {X 0,Y 356.336,Z 659.551,A -85,B 0,C 180,E1 -13514.226,E2 -13514.226} C_VEL
LIN {X 0,Y 355.788,Z 662.482,A -85,B 0,C 180,E1 -13516.055,E2 -13516.055} C_VEL
LIN {X 0,Y 355.281,Z 664.459,A -85,B 0,C 180,E1 -13518.288,E2 -13518.288} C_VEL
LIN {X 0,Y 355.118,Z 664.866,A -85,B 0,C 180,E1 -13519.661,E2 -13519.661} C_VEL
LIN {X 0,Y 354.962,Z 664.454,A -85,B 0,C 180,E1 -13521.48,E2 -13521.48} C_VEL
LIN {X 0,Y 354.926,Z 662.938,A -85,B 0,C 180,E1 -13523.33,E2 -13523.33} C_VEL
LIN {X 0,Y 355.132,Z 660.274,A -85,B 0,C 180,E1 -13525.182,E2 -13525.182} C_VEL
LIN {X 0,Y 355.403,Z 656.137,A -85,B 0,C 180,E1 -13527.147,E2 -13527.147} C_VEL
LIN {X 0,Y 355.761,Z 650.975,A -85,B 0,C 180,E1 -13528.947,E2 -13528.947} C_VEL
LIN {X 0,Y 356.309,Z 643.939,A -85,B 0,C 180,E1 -13530.853,E2 -13530.853} C_VEL
LIN {X 0,Y 356.902,Z 636.453,A -85,B 0,C 180,E1 -13532.453,E2 -13532.453} C_VEL
LIN {X 0,Y 357.536,Z 627.35,A -85,B 0,C 180,E1 -13534.026,E2 -13534.026} C_VEL
LIN {X 0,Y 358.259,Z 617.808,A -85,B 0,C 180,E1 -13535.36,E2 -13535.36} C_VEL
LIN {X 0,Y 358.861,Z 606.835,A -85,B 0,C 180,E1 -13536.589,E2 -13536.589} C_VEL
LIN {X 0,Y 359.459,Z 594.662,A -85,B 0,C 180,E1 -13537.662,E2 -13537.662} C_VEL
LIN {X 0,Y 359.819,Z 583.118,A -85,B 0,C 180,E1 -13538.432,E2 -13538.432} C_VEL
LIN {X 0,Y 360.07,Z 569.381,A -85,B 0,C 180,E1 -13539.089,E2 -13539.089} C_VEL
LIN {X 0,Y 360.108,Z 555.306,A -85,B 0,C 180,E1 -13539.496,E2 -13539.496} C_VEL
LIN {X 0,Y 360.011,Z 547.334,A -85,B 0,C 180,E1 -13539.684,E2 -13539.684} C_VEL
LIN {X 0,Y 355.03,Z 532.019,A -85,B 0,C 180,E1 -13540.265,E2 -13540.265} C_VEL
LIN {X 0,Y 354.853,Z 531.187,A -85,B 0,C 180,E1 -13540.476,E2 -13540.476} C_VEL
LIN {X 0,Y 354.814,Z 531.098,A -85,B 0,C 180,E1 -13544.516,E2 -13544.516} C_VEL
LIN {X 0,Y 354.836,Z 531.097,A -85,B 0,C 180,E1 -13547.67,E2 -13547.67} C_VEL
LIN {X 0,Y 354.837,Z 531.094,A -85,B 0,C 180,E1 -13550.67,E2 -13550.67} C_VEL
LIN {X 0,Y 354.822,Z 531.096,A -85,B 0,C 180,E1 -13554.302,E2 -13554.302} C_VEL
LIN {X 0,Y 354.787,Z 531.104,A -85,B 0,C 180,E1 -13557.668,E2 -13557.668} C_VEL
LIN {X 0,Y 354.87,Z 531.09,A -85,B 0,C 180,E1 -13560.622,E2 -13560.622} C_VEL
LIN {X 0,Y 354.902,Z 531.086,A -85,B 0,C 180,E1 -13564.174,E2 -13564.174} C_VEL
LIN {X 0,Y 354.838,Z 531.096,A -85,B 0,C 180,E1 -13567.895,E2 -13567.895} C_VEL
LIN {X 0,Y 354.893,Z 531.09,A -85,B 0,C 180,E1 -13571.908,E2 -13571.908} C_VEL
LIN {X 0,Y 354.947,Z 531.083,A -85,B 0,C 180,E1 -13575.982,E2 -13575.982} C_VEL
LIN {X 0,Y 354.982,Z 531.081,A -85,B 0,C 180,E1 -13579.736,E2 -13579.736} C_VEL
LIN {X 0,Y 355.104,Z 531.062,A -85,B 0,C 180,E1 -13583.18,E2 -13583.18} C_VEL
LIN {X 0,Y 355.248,Z 531.049,A -85,B 0,C 180,E1 -13587.733,E2 -13587.733} C_VEL
LIN {X 0,Y 355.401,Z 531.027,A -85,B 0,C 180,E1 -13590,E2 -13590} C_VEL
LIN {X 0,Y 355.248,Z 531.044,A -85,B 0,C 180,E1 -13592.268,E2 -13592.268} C_VEL
LIN {X 0,Y 355.104,Z 531.06,A -85,B 0,C 180,E1 -13596.82,E2 -13596.82} C_VEL
LIN {X 0,Y 354.961,Z 531.08,A -85,B 0,C 180,E1 -13600.264,E2 -13600.264} C_VEL
LIN {X 0,Y 354.947,Z 531.085,A -85,B 0,C 180,E1 -13604.019,E2 -13604.019} C_VEL
LIN {X 0,Y 354.927,Z 531.087,A -85,B 0,C 180,E1 -13608.108,E2 -13608.108} C_VEL
LIN {X 0,Y 354.818,Z 531.1,A -85,B 0,C 180,E1 -13612.107,E2 -13612.107} C_VEL
LIN {X 0,Y 354.9,Z 531.091,A -85,B 0,C 180,E1 -13615.827,E2 -13615.827} C_VEL
LIN {X 0,Y 354.819,Z 531.099,A -85,B 0,C 180,E1 -13619.681,E2 -13619.681} C_VEL
LIN {X 0,Y 354.807,Z 531.101,A -85,B 0,C 180,E1 -13623.701,E2 -13623.701} C_VEL
LIN {X 0,Y 354.804,Z 531.099,A -85,B 0,C 180,E1 -13626.072,E2 -13626.072} C_VEL
LIN {X 0,Y 354.123,Z 531.184,A -85,B 0,C 180,E1 -13627.019,E2 -13627.019} C_VEL
LIN {X 0,Y 351.268,Z 531.54,A -85,B 0,C 180,E1 -13628.56,E2 -13628.56} C_VEL
LIN {X 0,Y 348.865,Z 531.841,A -85,B 0,C 180,E1 -13629.807,E2 -13629.807} C_VEL
LIN {X 0,Y 347.845,Z 531.966,A -85,B 0,C 180,E1 -13630.772,E2 -13630.772} C_VEL
LIN {X 0,Y 347.767,Z 531.974,A -85,B 0,C 180,E1 -13631.099,E2 -13631.099} C_VEL
LIN {X 0,Y 347.796,Z 531.971,A -85,B 0,C 180,E1 -13634.987,E2 -13634.987} C_VEL
LIN {X 0,Y 347.749,Z 531.98,A -85,B 0,C 180,E1 -13638.396,E2 -13638.396} C_VEL
LIN {X 0,Y 347.772,Z 531.979,A -85,B 0,C 180,E1 -13642.01,E2 -13642.01} C_VEL
LIN {X 0,Y 347.741,Z 531.978,A -85,B 0,C 180,E1 -13645.535,E2 -13645.535} C_VEL
LIN {X 0,Y 347.762,Z 531.981,A -85,B 0,C 180,E1 -13648.302,E2 -13648.302} C_VEL
LIN {X 0,Y 347.803,Z 531.97,A -85,B 0,C 180,E1 -13650.989,E2 -13650.989} C_VEL
LIN {X 0,Y 347.827,Z 531.968,A -85,B 0,C 180,E1 -13653.607,E2 -13653.607} C_VEL
LIN {X 0,Y 347.784,Z 531.977,A -85,B 0,C 180,E1 -13656.161,E2 -13656.161} C_VEL
LIN {X 0,Y 347.822,Z 531.97,A -85,B 0,C 180,E1 -13659.909,E2 -13659.909} C_VEL
LIN {X 0,Y 347.861,Z 531.969,A -85,B 0,C 180,E1 -13662.359,E2 -13662.359} C_VEL
LIN {X 0,Y 347.892,Z 531.961,A -85,B 0,C 180,E1 -13665.97,E2 -13665.97} C_VEL
LIN {X 0,Y 347.926,Z 531.955,A -85,B 0,C 180,E1 -13669.525,E2 -13669.525} C_VEL
LIN {X 0,Y 348.068,Z 531.938,A -85,B 0,C 180,E1 -13671.874,E2 -13671.874} C_VEL
LIN {X 0,Y 348.062,Z 531.942,A -85,B 0,C 180,E1 -13674.205,E2 -13674.205} C_VEL
LIN {X 0,Y 348.201,Z 531.921,A -85,B 0,C 180,E1 -13677.686,E2 -13677.686} C_VEL
LIN {X 0,Y 348.338,Z 531.905,A -85,B 0,C 180,E1 -13680,E2 -13680} C_VEL
LIN {X 0,Y 348.201,Z 531.925,A -85,B 0,C 180,E1 -13682.313,E2 -13682.313} C_VEL
LIN {X 0,Y 348.085,Z 531.937,A -85,B 0,C 180,E1 -13686.958,E2 -13686.958} C_VEL
LIN {X 0,Y 347.921,Z 531.961,A -85,B 0,C 180,E1 -13690.474,E2 -13690.474} C_VEL
LIN {X 0,Y 347.891,Z 531.961,A -85,B 0,C 180,E1 -13694.15,E2 -13694.15} C_VEL
LIN {X 0,Y 347.884,Z 531.963,A -85,B 0,C 180,E1 -13698.29,E2 -13698.29} C_VEL
LIN {X 0,Y 347.761,Z 531.975,A -85,B 0,C 180,E1 -13701.626,E2 -13701.626} C_VEL
LIN {X 0,Y 347.804,Z 531.972,A -85,B 0,C 180,E1 -13705.109,E2 -13705.109} C_VEL
LIN {X 0,Y 347.806,Z 531.97,A -85,B 0,C 180,E1 -13707.694,E2 -13707.694} C_VEL
LIN {X 0,Y 347.758,Z 531.978,A -85,B 0,C 180,E1 -13710.347,E2 -13710.347} C_VEL
LIN {X 0,Y 347.738,Z 531.981,A -85,B 0,C 180,E1 -13714.464,E2 -13714.464} C_VEL
LIN {X 0,Y 347.768,Z 531.974,A -85,B 0,C 180,E1 -13717.989,E2 -13717.989} C_VEL
LIN {X 0,Y 347.745,Z 531.977,A -85,B 0,C 180,E1 -13721.831,E2 -13721.831} C_VEL
LIN {X 0,Y 347.762,Z 531.98,A -85,B 0,C 180,E1 -13725.017,E2 -13725.017} C_VEL
LIN {X 0,Y 347.747,Z 531.979,A -85,B 0,C 180,E1 -13728.398,E2 -13728.398} C_VEL
LIN {X 0,Y 347.771,Z 531.974,A -85,B 0,C 180,E1 -13732.012,E2 -13732.012} C_VEL
LIN {X 0,Y 347.872,Z 532.128,A -85,B 0,C 180,E1 -13735.376,E2 -13735.376} C_VEL
LIN {X 0,Y 350.773,Z 546.988,A -85,B 0,C 180,E1 -13739.489,E2 -13739.489} C_VEL
LIN {X 0,Y 351.481,Z 551.459,A -85,B 0,C 180,E1 -13740.668,E2 -13740.668} C_VEL
LIN {X 0,Y 350.2,Z 563.998,A -85,B 0,C 180,E1 -13743.8,E2 -13743.8} C_VEL
LIN {X 0,Y 348.738,Z 580.228,A -85,B 0,C 180,E1 -13747.81,E2 -13747.81} C_VEL
LIN {X 0,Y 347.752,Z 595.515,A -85,B 0,C 180,E1 -13751.561,E2 -13751.561} C_VEL
LIN {X 0,Y 347.661,Z 597.166,A -85,B 0,C 180,E1 -13751.876,E2 -13751.876} C_VEL
LIN {X 0,Y 351.673,Z 648.97,A -85,B 0,C 180,E1 -13753.473,E2 -13753.473} C_VEL
LIN {X 0,Y 350.942,Z 681.559,A -85,B 0,C 180,E1 -13754.379,E2 -13754.379} C_VEL
LIN {X 0,Y 350.414,Z 693.945,A -85,B 0,C 180,E1 -13754.961,E2 -13754.961} C_VEL
LIN {X 0,Y 349.496,Z 705.457,A -85,B 0,C 180,E1 -13755.74,E2 -13755.74} C_VEL
LIN {X 0,Y 348.804,Z 716.443,A -85,B 0,C 180,E1 -13756.751,E2 -13756.751} C_VEL
LIN {X 0,Y 348.005,Z 726.2,A -85,B 0,C 180,E1 -13757.906,E2 -13757.906} C_VEL
LIN {X 0,Y 347.384,Z 734.982,A -85,B 0,C 180,E1 -13759.214,E2 -13759.214} C_VEL
LIN {X 0,Y 347.031,Z 742.76,A -85,B 0,C 180,E1 -13760.676,E2 -13760.676} C_VEL
LIN {X 0,Y 346.915,Z 749.006,A -85,B 0,C 180,E1 -13762.141,E2 -13762.141} C_VEL
LIN {X 0,Y 346.928,Z 754.53,A -85,B 0,C 180,E1 -13763.807,E2 -13763.807} C_VEL
LIN {X 0,Y 347.08,Z 758.398,A -85,B 0,C 180,E1 -13765.354,E2 -13765.354} C_VEL
LIN {X 0,Y 347.208,Z 760.583,A -85,B 0,C 180,E1 -13766.519,E2 -13766.519} C_VEL
LIN {X 0,Y 347.287,Z 762.148,A -85,B 0,C 180,E1 -13767.68,E2 -13767.68} C_VEL
LIN {X 0,Y 347.404,Z 763.15,A -85,B 0,C 180,E1 -13768.841,E2 -13768.841} C_VEL
LIN {X 0,Y 347.651,Z 763.63,A -85,B 0,C 180,E1 -13770,E2 -13770} C_VEL
LIN {X 0,Y 347.33,Z 763.456,A -85,B 0,C 180,E1 -13771.159,E2 -13771.159} C_VEL
LIN {X 0,Y 347.203,Z 762.792,A -85,B 0,C 180,E1 -13772.32,E2 -13772.32} C_VEL
LIN {X 0,Y 347.147,Z 761.566,A -85,B 0,C 180,E1 -13773.482,E2 -13773.482} C_VEL
LIN {X 0,Y 346.842,Z 758.68,A -85,B 0,C 180,E1 -13775.231,E2 -13775.231} C_VEL
LIN {X 0,Y 346.696,Z 754.469,A -85,B 0,C 180,E1 -13776.986,E2 -13776.986} C_VEL
LIN {X 0,Y 346.852,Z 748.847,A -85,B 0,C 180,E1 -13778.741,E2 -13778.741} C_VEL
LIN {X 0,Y 347.149,Z 742.912,A -85,B 0,C 180,E1 -13780.203,E2 -13780.203} C_VEL
LIN {X 0,Y 347.704,Z 735.573,A -85,B 0,C 180,E1 -13781.661,E2 -13781.661} C_VEL
LIN {X 0,Y 348.707,Z 726.543,A -85,B 0,C 180,E1 -13783.105,E2 -13783.105} C_VEL
LIN {X 0,Y 349.89,Z 716.326,A -85,B 0,C 180,E1 -13784.392,E2 -13784.392} C_VEL
LIN {X 0,Y 350.968,Z 706.402,A -85,B 0,C 180,E1 -13785.386,E2 -13785.386} C_VEL
LIN {X 0,Y 352.224,Z 693.796,A -85,B 0,C 180,E1 -13786.351,E2 -13786.351} C_VEL
LIN {X 0,Y 353.355,Z 680.349,A -85,B 0,C 180,E1 -13787.079,E2 -13787.079} C_VEL
LIN {X 0,Y 353.961,Z 666.793,A -85,B 0,C 180,E1 -13787.55,E2 -13787.55} C_VEL
LIN {X 0,Y 354.291,Z 646.952,A -85,B 0,C 180,E1 -13788.074,E2 -13788.074} C_VEL
LIN {X 0,Y 352.905,Z 621.316,A -85,B 0,C 180,E1 -13788.899,E2 -13788.899} C_VEL
LIN {X 0,Y 350.725,Z 601.404,A -85,B 0,C 180,E1 -13789.643,E2 -13789.643} C_VEL
LIN {X 0,Y 347.964,Z 584.151,A -85,B 0,C 180,E1 -13790.428,E2 -13790.428} C_VEL
LIN {X 0,Y 348.526,Z 575.27,A -85,B 0,C 180,E1 -13792.527,E2 -13792.527} C_VEL
LIN {X 0,Y 349.875,Z 559.223,A -85,B 0,C 180,E1 -13796.547,E2 -13796.547} C_VEL
LIN {X 0,Y 350.882,Z 549.564,A -85,B 0,C 180,E1 -13799.059,E2 -13799.059} C_VEL
LIN {X 0,Y 350.344,Z 544.817,A -85,B 0,C 180,E1 -13800.392,E2 -13800.392} C_VEL
LIN {X 0,Y 348.334,Z 534.461,A -85,B 0,C 180,E1 -13803.529,E2 -13803.529} C_VEL
LIN {X 0,Y 347.824,Z 532.008,A -85,B 0,C 180,E1 -13804.392,E2 -13804.392} C_VEL
LIN {X 0,Y 347.77,Z 531.978,A -85,B 0,C 180,E1 -13807.988,E2 -13807.988} C_VEL
LIN {X 0,Y 347.746,Z 531.979,A -85,B 0,C 180,E1 -13811.83,E2 -13811.83} C_VEL
LIN {X 0,Y 347.792,Z 531.971,A -85,B 0,C 180,E1 -13815.011,E2 -13815.011} C_VEL
LIN {X 0,Y 347.778,Z 531.97,A -85,B 0,C 180,E1 -13818.39,E2 -13818.39} C_VEL
LIN {X 0,Y 347.775,Z 531.975,A -85,B 0,C 180,E1 -13822.009,E2 -13822.009} C_VEL
LIN {X 0,Y 347.738,Z 531.982,A -85,B 0,C 180,E1 -13825.536,E2 -13825.536} C_VEL
LIN {X 0,Y 347.757,Z 531.976,A -85,B 0,C 180,E1 -13828.302,E2 -13828.302} C_VEL
LIN {X 0,Y 347.799,Z 531.97,A -85,B 0,C 180,E1 -13830.99,E2 -13830.99} C_VEL
LIN {X 0,Y 347.824,Z 531.964,A -85,B 0,C 180,E1 -13833.608,E2 -13833.608} C_VEL
LIN {X 0,Y 347.781,Z 531.974,A -85,B 0,C 180,E1 -13836.162,E2 -13836.162} C_VEL
LIN {X 0,Y 347.804,Z 531.969,A -85,B 0,C 180,E1 -13839.909,E2 -13839.909} C_VEL
LIN {X 0,Y 347.858,Z 531.963,A -85,B 0,C 180,E1 -13842.359,E2 -13842.359} C_VEL
LIN {X 0,Y 347.889,Z 531.963,A -85,B 0,C 180,E1 -13845.971,E2 -13845.971} C_VEL
LIN {X 0,Y 347.925,Z 531.959,A -85,B 0,C 180,E1 -13849.526,E2 -13849.526} C_VEL
LIN {X 0,Y 348.066,Z 531.943,A -85,B 0,C 180,E1 -13851.875,E2 -13851.875} C_VEL
LIN {X 0,Y 348.065,Z 531.942,A -85,B 0,C 180,E1 -13854.206,E2 -13854.206} C_VEL
LIN {X 0,Y 348.201,Z 531.927,A -85,B 0,C 180,E1 -13857.687,E2 -13857.687} C_VEL
LIN {X 0,Y 348.194,Z 532.163,A -85,B 0,C 180,E1 -13859.024,E2 -13859.024} C_VEL
LIN {X 0,Y 348.514,Z 533.374,A -85,B 0,C 180,E1 -13859.231,E2 -13859.231} C_VEL
LIN {X 0,Y 351.858,Z 540.025,A -85,B 0,C 180,E1 -13859.705,E2 -13859.705} C_VEL
LIN {X 0,Y 356.96,Z 551.749,A -85,B 0,C 180,E1 -13860.421,E2 -13860.421} C_VEL
LIN {X 0,Y 357.129,Z 573.54,A -85,B 0,C 180,E1 -13861.012,E2 -13861.012} C_VEL
LIN {X 0,Y 357.005,Z 586.155,A -85,B 0,C 180,E1 -13861.584,E2 -13861.584} C_VEL
LIN {X 0,Y 356.615,Z 596.739,A -85,B 0,C 180,E1 -13862.259,E2 -13862.259} C_VEL
LIN {X 0,Y 355.799,Z 608.66,A -85,B 0,C 180,E1 -13863.256,E2 -13863.256} C_VEL
LIN {X 0,Y 354.992,Z 619.238,A -85,B 0,C 180,E1 -13864.4,E2 -13864.4} C_VEL
LIN {X 0,Y 354.036,Z 628.764,A -85,B 0,C 180,E1 -13865.697,E2 -13865.697} C_VEL
LIN {X 0,Y 353.016,Z 637.387,A -85,B 0,C 180,E1 -13867.148,E2 -13867.148} C_VEL
LIN {X 0,Y 352.08,Z 644.432,A -85,B 0,C 180,E1 -13868.611,E2 -13868.611} C_VEL
LIN {X 0,Y 351.04,Z 651.221,A -85,B 0,C 180,E1 -13870.381,E2 -13870.381} C_VEL
LIN {X 0,Y 350.213,Z 656.517,A -85,B 0,C 180,E1 -13872.165,E2 -13872.165} C_VEL
LIN {X 0,Y 349.443,Z 660.576,A -85,B 0,C 180,E1 -13873.966,E2 -13873.966} C_VEL
LIN {X 0,Y 349.033,Z 662.611,A -85,B 0,C 180,E1 -13875.175,E2 -13875.175} C_VEL
LIN {X 0,Y 348.688,Z 664.153,A -85,B 0,C 180,E1 -13876.391,E2 -13876.391} C_VEL
LIN {X 0,Y 348.263,Z 665.702,A -85,B 0,C 180,E1 -13878.478,E2 -13878.478} C_VEL
LIN {X 0,Y 348.07,Z 665.928,A -85,B 0,C 180,E1 -13880.076,E2 -13880.076} C_VEL
LIN {X 0,Y 347.918,Z 665.343,A -85,B 0,C 180,E1 -13881.692,E2 -13881.692} C_VEL
LIN {X 0,Y 347.934,Z 663.33,A -85,B 0,C 180,E1 -13883.828,E2 -13883.828} C_VEL
LIN {X 0,Y 348.135,Z 660.272,A -85,B 0,C 180,E1 -13885.724,E2 -13885.724} C_VEL
LIN {X 0,Y 348.449,Z 655.922,A -85,B 0,C 180,E1 -13887.639,E2 -13887.639} C_VEL
LIN {X 0,Y 348.851,Z 650.416,A -85,B 0,C 180,E1 -13889.477,E2 -13889.477} C_VEL
LIN {X 0,Y 349.384,Z 643.816,A -85,B 0,C 180,E1 -13891.197,E2 -13891.197} C_VEL
LIN {X 0,Y 350.036,Z 636.049,A -85,B 0,C 180,E1 -13892.828,E2 -13892.828} C_VEL
LIN {X 0,Y 350.662,Z 627.018,A -85,B 0,C 180,E1 -13894.372,E2 -13894.372} C_VEL
LIN {X 0,Y 351.397,Z 616.497,A -85,B 0,C 180,E1 -13895.804,E2 -13895.804} C_VEL
LIN {X 0,Y 352.018,Z 605.509,A -85,B 0,C 180,E1 -13897.006,E2 -13897.006} C_VEL
LIN {X 0,Y 352.62,Z 593.913,A -85,B 0,C 180,E1 -13897.991,E2 -13897.991} C_VEL
LIN {X 0,Y 352.983,Z 582.001,A -85,B 0,C 180,E1 -13898.767,E2 -13898.767} C_VEL
LIN {X 0,Y 353.158,Z 569.184,A -85,B 0,C 180,E1 -13899.362,E2 -13899.362} C_VEL
LIN {X 0,Y 353.201,Z 551.661,A -85,B 0,C 180,E1 -13899.846,E2 -13899.846} C_VEL
LIN {X 0,Y 353.103,Z 548.568,A -85,B 0,C 180,E1 -13899.924,E2 -13899.924} C_VEL
LIN {X 0,Y 348.027,Z 533.056,A -85,B 0,C 180,E1 -13900.526,E2 -13900.526} C_VEL
LIN {X 0,Y 347.778,Z 532.099,A -85,B 0,C 180,E1 -13900.737,E2 -13900.737} C_VEL
LIN {X 0,Y 347.796,Z 531.974,A -85,B 0,C 180,E1 -13905.013,E2 -13905.013} C_VEL
LIN {X 0,Y 347.783,Z 531.972,A -85,B 0,C 180,E1 -13908.392,E2 -13908.392} C_VEL
LIN {X 0,Y 347.776,Z 531.974,A -85,B 0,C 180,E1 -13912.012,E2 -13912.012} C_VEL
LIN {X 0,Y 347.745,Z 531.983,A -85,B 0,C 180,E1 -13915.537,E2 -13915.537} C_VEL
LIN {X 0,Y 347.765,Z 531.979,A -85,B 0,C 180,E1 -13919.655,E2 -13919.655} C_VEL
LIN {X 0,Y 347.853,Z 531.964,A -85,B 0,C 180,E1 -13922.746,E2 -13922.746} C_VEL
LIN {X 0,Y 347.791,Z 531.972,A -85,B 0,C 180,E1 -13926.163,E2 -13926.163} C_VEL
LIN {X 0,Y 347.809,Z 531.972,A -85,B 0,C 180,E1 -13929.91,E2 -13929.91} C_VEL
LIN {X 0,Y 347.836,Z 531.972,A -85,B 0,C 180,E1 -13933.569,E2 -13933.569} C_VEL
LIN {X 0,Y 347.894,Z 531.96,A -85,B 0,C 180,E1 -13937.161,E2 -13937.161} C_VEL
LIN {X 0,Y 347.946,Z 531.952,A -85,B 0,C 180,E1 -13940.701,E2 -13940.701} C_VEL
LIN {X 0,Y 348.054,Z 531.94,A -85,B 0,C 180,E1 -13944.206,E2 -13944.206} C_VEL
LIN {X 0,Y 348.21,Z 531.925,A -85,B 0,C 180,E1 -13947.687,E2 -13947.687} C_VEL
LIN {X 0,Y 348.349,Z 531.905,A -85,B 0,C 180,E1 -13950,E2 -13950} C_VEL
LIN {X 0,Y 348.211,Z 531.92,A -85,B 0,C 180,E1 -13952.313,E2 -13952.313} C_VEL
LIN {X 0,Y 348.072,Z 531.937,A -85,B 0,C 180,E1 -13956.958,E2 -13956.958} C_VEL
LIN {X 0,Y 347.901,Z 531.958,A -85,B 0,C 180,E1 -13960.475,E2 -13960.475} C_VEL
LIN {X 0,Y 347.902,Z 531.961,A -85,B 0,C 180,E1 -13964.149,E2 -13964.149} C_VEL
LIN {X 0,Y 347.895,Z 531.961,A -85,B 0,C 180,E1 -13968.29,E2 -13968.29} C_VEL
LIN {X 0,Y 347.771,Z 531.977,A -85,B 0,C 180,E1 -13971.626,E2 -13971.626} C_VEL
LIN {X 0,Y 347.813,Z 531.969,A -85,B 0,C 180,E1 -13975.108,E2 -13975.108} C_VEL
LIN {X 0,Y 347.81,Z 531.973,A -85,B 0,C 180,E1 -13977.693,E2 -13977.693} C_VEL
LIN {X 0,Y 347.751,Z 531.979,A -85,B 0,C 180,E1 -13980.347,E2 -13980.347} C_VEL
LIN {X 0,Y 347.749,Z 531.983,A -85,B 0,C 180,E1 -13984.043,E2 -13984.043} C_VEL
LIN {X 0,Y 347.763,Z 531.975,A -85,B 0,C 180,E1 -13987.32,E2 -13987.32} C_VEL
LIN {X 0,Y 347.767,Z 531.974,A -85,B 0,C 180,E1 -13991.099,E2 -13991.099} C_VEL
LIN {X 0,Y 347.114,Z 532.062,A -85,B 0,C 180,E1 -13992.066,E2 -13992.066} C_VEL
LIN {X 0,Y 344.264,Z 532.422,A -85,B 0,C 180,E1 -13993.639,E2 -13993.639} C_VEL
LIN {X 0,Y 341.83,Z 532.728,A -85,B 0,C 180,E1 -13994.913,E2 -13994.913} C_VEL
LIN {X 0,Y 340.769,Z 532.855,A -85,B 0,C 180,E1 -13995.898,E2 -13995.898} C_VEL
LIN {X 0,Y 340.675,Z 532.863,A -85,B 0,C 180,E1 -13996.232,E2 -13996.232} C_VEL
LIN {X 0,Y 340.686,Z 532.859,A -85,B 0,C 180,E1 -13999.752,E2 -13999.752} C_VEL
LIN {X 0,Y 340.703,Z 532.854,A -85,B 0,C 180,E1 -14003.257,E2 -14003.257} C_VEL
LIN {X 0,Y 340.692,Z 532.862,A -85,B 0,C 180,E1 -14006.153,E2 -14006.153} C_VEL
LIN {X 0,Y 340.772,Z 532.851,A -85,B 0,C 180,E1 -14010.332,E2 -14010.332} C_VEL
LIN {X 0,Y 340.801,Z 532.843,A -85,B 0,C 180,E1 -14013.019,E2 -14013.019} C_VEL
LIN {X 0,Y 340.725,Z 532.852,A -85,B 0,C 180,E1 -14016.926,E2 -14016.926} C_VEL
LIN {X 0,Y 340.794,Z 532.845,A -85,B 0,C 180,E1 -14020.733,E2 -14020.733} C_VEL
LIN {X 0,Y 340.781,Z 532.845,A -85,B 0,C 180,E1 -14023.218,E2 -14023.218} C_VEL
LIN {X 0,Y 340.84,Z 532.839,A -85,B 0,C 180,E1 -14026.89,E2 -14026.89} C_VEL
LIN {X 0,Y 340.924,Z 532.832,A -85,B 0,C 180,E1 -14030.507,E2 -14030.507} C_VEL
LIN {X 0,Y 341.07,Z 532.811,A -85,B 0,C 180,E1 -14032.898,E2 -14032.898} C_VEL
LIN {X 0,Y 341.163,Z 532.797,A -85,B 0,C 180,E1 -14037.638,E2 -14037.638} C_VEL
LIN {X 0,Y 341.289,Z 532.783,A -85,B 0,C 180,E1 -14040,E2 -14040} C_VEL
LIN {X 0,Y 341.163,Z 532.802,A -85,B 0,C 180,E1 -14042.361,E2 -14042.361} C_VEL
LIN {X 0,Y 341.054,Z 532.812,A -85,B 0,C 180,E1 -14047.102,E2 -14047.102} C_VEL
LIN {X 0,Y 340.863,Z 532.84,A -85,B 0,C 180,E1 -14050.694,E2 -14050.694} C_VEL
LIN {X 0,Y 340.856,Z 532.839,A -85,B 0,C 180,E1 -14054.325,E2 -14054.325} C_VEL
LIN {X 0,Y 340.831,Z 532.843,A -85,B 0,C 180,E1 -14058.467,E2 -14058.467} C_VEL
LIN {X 0,Y 340.711,Z 532.854,A -85,B 0,C 180,E1 -14061.842,E2 -14061.842} C_VEL
LIN {X 0,Y 340.765,Z 532.847,A -85,B 0,C 180,E1 -14065.665,E2 -14065.665} C_VEL
LIN {X 0,Y 340.736,Z 532.853,A -85,B 0,C 180,E1 -14068.32,E2 -14068.32} C_VEL
LIN {X 0,Y 340.698,Z 532.858,A -85,B 0,C 180,E1 -14071.044,E2 -14071.044} C_VEL
LIN {X 0,Y 340.712,Z 532.855,A -85,B 0,C 180,E1 -14075.279,E2 -14075.279} C_VEL
LIN {X 0,Y 340.704,Z 532.856,A -85,B 0,C 180,E1 -14078.386,E2 -14078.386} C_VEL
LIN {X 0,Y 340.694,Z 532.856,A -85,B 0,C 180,E1 -14082.046,E2 -14082.046} C_VEL
LIN {X 0,Y 340.679,Z 532.858,A -85,B 0,C 180,E1 -14085.462,E2 -14085.462} C_VEL
LIN {X 0,Y 340.682,Z 532.861,A -85,B 0,C 180,E1 -14088.691,E2 -14088.691} C_VEL
LIN {X 0,Y 340.73,Z 532.851,A -85,B 0,C 180,E1 -14091.773,E2 -14091.773} C_VEL
LIN {X 0,Y 340.818,Z 533.015,A -85,B 0,C 180,E1 -14095.185,E2 -14095.185} C_VEL
LIN {X 0,Y 343.618,Z 547.352,A -85,B 0,C 180,E1 -14099.249,E2 -14099.249} C_VEL
LIN {X 0,Y 344.433,Z 552.655,A -85,B 0,C 180,E1 -14100.679,E2 -14100.679} C_VEL
LIN {X 0,Y 342.875,Z 567.628,A -85,B 0,C 180,E1 -14104.505,E2 -14104.505} C_VEL
LIN {X 0,Y 341.32,Z 584.943,A -85,B 0,C 180,E1 -14108.88,E2 -14108.88} C_VEL
LIN {X 0,Y 340.675,Z 595.641,A -85,B 0,C 180,E1 -14111.532,E2 -14111.532} C_VEL
LIN {X 0,Y 341.089,Z 603,A -85,B 0,C 180,E1 -14111.809,E2 -14111.809} C_VEL
LIN {X 0,Y 344.692,Z 649.713,A -85,B 0,C 180,E1 -14113.262,E2 -14113.262} C_VEL
LIN {X 0,Y 343.971,Z 680.615,A -85,B 0,C 180,E1 -14114.153,E2 -14114.153} C_VEL
LIN {X 0,Y 343.48,Z 692.569,A -85,B 0,C 180,E1 -14114.726,E2 -14114.726} C_VEL
LIN {X 0,Y 342.612,Z 703.2,A -85,B 0,C 180,E1 -14115.447,E2 -14115.447} C_VEL
LIN {X 0,Y 342.007,Z 713.079,A -85,B 0,C 180,E1 -14116.331,E2 -14116.331} C_VEL
LIN {X 0,Y 341.177,Z 723.343,A -85,B 0,C 180,E1 -14117.509,E2 -14117.509} C_VEL
LIN {X 0,Y 340.493,Z 731.543,A -85,B 0,C 180,E1 -14118.692,E2 -14118.692} C_VEL
LIN {X 0,Y 340.056,Z 739.837,A -85,B 0,C 180,E1 -14120.183,E2 -14120.183} C_VEL
LIN {X 0,Y 339.848,Z 746.448,A -85,B 0,C 180,E1 -14121.677,E2 -14121.677} C_VEL
LIN {X 0,Y 339.888,Z 752.383,A -85,B 0,C 180,E1 -14123.387,E2 -14123.387} C_VEL
LIN {X 0,Y 340.027,Z 757.169,A -85,B 0,C 180,E1 -14125.258,E2 -14125.258} C_VEL
LIN {X 0,Y 340.166,Z 759.412,A -85,B 0,C 180,E1 -14126.446,E2 -14126.446} C_VEL
LIN {X 0,Y 340.254,Z 761.008,A -85,B 0,C 180,E1 -14127.632,E2 -14127.632} C_VEL
LIN {X 0,Y 340.399,Z 762.069,A -85,B 0,C 180,E1 -14128.817,E2 -14128.817} C_VEL
LIN {X 0,Y 340.643,Z 762.57,A -85,B 0,C 180,E1 -14130,E2 -14130} C_VEL
LIN {X 0,Y 340.292,Z 762.441,A -85,B 0,C 180,E1 -14131.183,E2 -14131.183} C_VEL
LIN {X 0,Y 340.156,Z 761.795,A -85,B 0,C 180,E1 -14132.368,E2 -14132.368} C_VEL
LIN {X 0,Y 340.095,Z 760.609,A -85,B 0,C 180,E1 -14133.554,E2 -14133.554} C_VEL
LIN {X 0,Y 339.762,Z 757.773,A -85,B 0,C 180,E1 -14135.341,E2 -14135.341} C_VEL
LIN {X 0,Y 339.63,Z 753.659,A -85,B 0,C 180,E1 -14137.132,E2 -14137.132} C_VEL
LIN {X 0,Y 339.78,Z 748.098,A -85,B 0,C 180,E1 -14138.924,E2 -14138.924} C_VEL
LIN {X 0,Y 340.212,Z 740.906,A -85,B 0,C 180,E1 -14140.714,E2 -14140.714} C_VEL
LIN {X 0,Y 340.908,Z 733.373,A -85,B 0,C 180,E1 -14142.199,E2 -14142.199} C_VEL
LIN {X 0,Y 342.041,Z 724.061,A -85,B 0,C 180,E1 -14143.667,E2 -14143.667} C_VEL
LIN {X 0,Y 343.263,Z 713.615,A -85,B 0,C 180,E1 -14144.98,E2 -14144.98} C_VEL
LIN {X 0,Y 344.732,Z 701.706,A -85,B 0,C 180,E1 -14146.127,E2 -14146.127} C_VEL
LIN {X 0,Y 345.921,Z 689.627,A -85,B 0,C 180,E1 -14146.998,E2 -14146.998} C_VEL
LIN {X 0,Y 346.85,Z 677.726,A -85,B 0,C 180,E1 -14147.617,E2 -14147.617} C_VEL
LIN {X 0,Y 347.515,Z 664.598,A -85,B 0,C 180,E1 -14148.062,E2 -14148.062} C_VEL
LIN {X 0,Y 347.799,Z 647.813,A -85,B 0,C 180,E1 -14148.519,E2 -14148.519} C_VEL
LIN {X 0,Y 346.4,Z 620.869,A -85,B 0,C 180,E1 -14149.414,E2 -14149.414} C_VEL
LIN {X 0,Y 344.093,Z 600.46,A -85,B 0,C 180,E1 -14150.226,E2 -14150.226} C_VEL
LIN {X 0,Y 341.081,Z 582.453,A -85,B 0,C 180,E1 -14151.083,E2 -14151.083} C_VEL
LIN {X 0,Y 341.21,Z 579.364,A -85,B 0,C 180,E1 -14151.761,E2 -14151.761} C_VEL
LIN {X 0,Y 342.452,Z 564.555,A -85,B 0,C 180,E1 -14155.529,E2 -14155.529} C_VEL
LIN {X 0,Y 343.816,Z 552.053,A -85,B 0,C 180,E1 -14158.821,E2 -14158.821} C_VEL
LIN {X 0,Y 343.831,Z 548.849,A -85,B 0,C 180,E1 -14159.713,E2 -14159.713} C_VEL
LIN {X 0,Y 342.08,Z 539.299,A -85,B 0,C 180,E1 -14162.612,E2 -14162.612} C_VEL
LIN {X 0,Y 340.781,Z 532.904,A -85,B 0,C 180,E1 -14164.76,E2 -14164.76} C_VEL
LIN {X 0,Y 340.706,Z 532.857,A -85,B 0,C 180,E1 -14168.386,E2 -14168.386} C_VEL
LIN {X 0,Y 340.695,Z 532.856,A -85,B 0,C 180,E1 -14172.045,E2 -14172.045} C_VEL
LIN {X 0,Y 340.716,Z 532.854,A -85,B 0,C 180,E1 -14175.467,E2 -14175.467} C_VEL
LIN {X 0,Y 340.72,Z 532.852,A -85,B 0,C 180,E1 -14178.696,E2 -14178.696} C_VEL
LIN {X 0,Y 340.74,Z 532.852,A -85,B 0,C 180,E1 -14181.774,E2 -14181.774} C_VEL
LIN {X 0,Y 340.716,Z 532.857,A -85,B 0,C 180,E1 -14185.595,E2 -14185.595} C_VEL
LIN {X 0,Y 340.709,Z 532.86,A -85,B 0,C 180,E1 -14188.957,E2 -14188.957} C_VEL
LIN {X 0,Y 340.773,Z 532.851,A -85,B 0,C 180,E1 -14192.474,E2 -14192.474} C_VEL
LIN {X 0,Y 340.748,Z 532.851,A -85,B 0,C 180,E1 -14195.638,E2 -14195.638} C_VEL
LIN {X 0,Y 340.737,Z 532.849,A -85,B 0,C 180,E1 -14199.474,E2 -14199.474} C_VEL
LIN {X 0,Y 340.849,Z 532.836,A -85,B 0,C 180,E1 -14201.984,E2 -14201.984} C_VEL
LIN {X 0,Y 340.861,Z 532.839,A -85,B 0,C 180,E1 -14205.705,E2 -14205.705} C_VEL
LIN {X 0,Y 340.867,Z 532.837,A -85,B 0,C 180,E1 -14209.307,E2 -14209.307} C_VEL
LIN {X 0,Y 341.07,Z 532.813,A -85,B 0,C 180,E1 -14212.899,E2 -14212.899} C_VEL
LIN {X 0,Y 341.163,Z 532.804,A -85,B 0,C 180,E1 -14217.639,E2 -14217.639} C_VEL
LIN {X 0,Y 341.144,Z 533.053,A -85,B 0,C 180,E1 -14218.377,E2 -14218.377} C_VEL
LIN {X 0,Y 341.357,Z 534.031,A -85,B 0,C 180,E1 -14218.563,E2 -14218.563} C_VEL
LIN {X 0,Y 346.101,Z 543.251,A -85,B 0,C 180,E1 -14219.281,E2 -14219.281} C_VEL
LIN {X 0,Y 350.736,Z 553.903,A -85,B 0,C 180,E1 -14219.965,E2 -14219.965} C_VEL
LIN {X 0,Y 350.777,Z 575.276,A -85,B 0,C 180,E1 -14220.556,E2 -14220.556} C_VEL
LIN {X 0,Y 350.648,Z 586.373,A -85,B 0,C 180,E1 -14221.066,E2 -14221.066} C_VEL
LIN {X 0,Y 350.248,Z 596.889,A -85,B 0,C 180,E1 -14221.725,E2 -14221.725} C_VEL
LIN {X 0,Y 349.56,Z 607.519,A -85,B 0,C 180,E1 -14222.593,E2 -14222.593} C_VEL
LIN {X 0,Y 348.659,Z 618.526,A -85,B 0,C 180,E1 -14223.757,E2 -14223.757} C_VEL
LIN {X 0,Y 347.745,Z 627.425,A -85,B 0,C 180,E1 -14224.928,E2 -14224.928} C_VEL
LIN {X 0,Y 346.572,Z 636.871,A -85,B 0,C 180,E1 -14226.473,E2 -14226.473} C_VEL
LIN {X 0,Y 345.43,Z 645.195,A -85,B 0,C 180,E1 -14228.188,E2 -14228.188} C_VEL
LIN {X 0,Y 344.339,Z 652.078,A -85,B 0,C 180,E1 -14229.991,E2 -14229.991} C_VEL
LIN {X 0,Y 343.431,Z 657.434,A -85,B 0,C 180,E1 -14231.809,E2 -14231.809} C_VEL
LIN {X 0,Y 342.607,Z 661.537,A -85,B 0,C 180,E1 -14233.645,E2 -14233.645} C_VEL
LIN {X 0,Y 341.944,Z 664.462,A -85,B 0,C 180,E1 -14235.498,E2 -14235.498} C_VEL
LIN {X 0,Y 341.602,Z 665.776,A -85,B 0,C 180,E1 -14236.741,E2 -14236.741} C_VEL
LIN {X 0,Y 341.225,Z 666.87,A -85,B 0,C 180,E1 -14238.665,E2 -14238.665} C_VEL
LIN {X 0,Y 341,Z 666.871,A -85,B 0,C 180,E1 -14240.51,E2 -14240.51} C_VEL
LIN {X 0,Y 340.878,Z 666.216,A -85,B 0,C 180,E1 -14241.912,E2 -14241.912} C_VEL
LIN {X 0,Y 340.856,Z 665.191,A -85,B 0,C 180,E1 -14243.064,E2 -14243.064} C_VEL
LIN {X 0,Y 341.032,Z 662.657,A -85,B 0,C 180,E1 -14244.943,E2 -14244.943} C_VEL
LIN {X 0,Y 341.294,Z 658.726,A -85,B 0,C 180,E1 -14246.939,E2 -14246.939} C_VEL
LIN {X 0,Y 341.663,Z 653.421,A -85,B 0,C 180,E1 -14248.908,E2 -14248.908} C_VEL
LIN {X 0,Y 342.238,Z 646.436,A -85,B 0,C 180,E1 -14250.89,E2 -14250.89} C_VEL
LIN {X 0,Y 342.842,Z 639.159,A -85,B 0,C 180,E1 -14252.535,E2 -14252.535} C_VEL
LIN {X 0,Y 343.556,Z 629.761,A -85,B 0,C 180,E1 -14254.233,E2 -14254.233} C_VEL
LIN {X 0,Y 344.324,Z 619.895,A -85,B 0,C 180,E1 -14255.672,E2 -14255.672} C_VEL
LIN {X 0,Y 344.953,Z 608.964,A -85,B 0,C 180,E1 -14256.944,E2 -14256.944} C_VEL
LIN {X 0,Y 345.618,Z 596.844,A -85,B 0,C 180,E1 -14258.054,E2 -14258.054} C_VEL
LIN {X 0,Y 345.997,Z 584.018,A -85,B 0,C 180,E1 -14258.934,E2 -14258.934} C_VEL
LIN {X 0,Y 346.252,Z 570.863,A -85,B 0,C 180,E1 -14259.573,E2 -14259.573} C_VEL
LIN {X 0,Y 346.283,Z 553.628,A -85,B 0,C 180,E1 -14260.067,E2 -14260.067} C_VEL
LIN {X 0,Y 346.172,Z 549.797,A -85,B 0,C 180,E1 -14260.166,E2 -14260.166} C_VEL
LIN {X 0,Y 340.918,Z 533.826,A -85,B 0,C 180,E1 -14260.801,E2 -14260.801} C_VEL
LIN {X 0,Y 340.72,Z 532.947,A -85,B 0,C 180,E1 -14261.025,E2 -14261.025} C_VEL
LIN {X 0,Y 340.703,Z 532.857,A -85,B 0,C 180,E1 -14264.536,E2 -14264.536} C_VEL
LIN {X 0,Y 340.746,Z 532.85,A -85,B 0,C 180,E1 -14267.947,E2 -14267.947} C_VEL
LIN {X 0,Y 340.734,Z 532.851,A -85,B 0,C 180,E1 -14270.254,E2 -14270.254} C_VEL
LIN {X 0,Y 340.711,Z 532.858,A -85,B 0,C 180,E1 -14273.56,E2 -14273.56} C_VEL
LIN {X 0,Y 340.692,Z 532.856,A -85,B 0,C 180,E1 -14276.154,E2 -14276.154} C_VEL
LIN {X 0,Y 340.776,Z 532.845,A -85,B 0,C 180,E1 -14280.333,E2 -14280.333} C_VEL
LIN {X 0,Y 340.807,Z 532.843,A -85,B 0,C 180,E1 -14283.021,E2 -14283.021} C_VEL
LIN {X 0,Y 340.731,Z 532.852,A -85,B 0,C 180,E1 -14286.928,E2 -14286.928} C_VEL
LIN {X 0,Y 340.763,Z 532.847,A -85,B 0,C 180,E1 -14290.732,E2 -14290.732} C_VEL
LIN {X 0,Y 340.821,Z 532.84,A -85,B 0,C 180,E1 -14294.451,E2 -14294.451} C_VEL
LIN {X 0,Y 340.854,Z 532.838,A -85,B 0,C 180,E1 -14298.101,E2 -14298.101} C_VEL
LIN {X 0,Y 340.983,Z 532.826,A -85,B 0,C 180,E1 -14301.705,E2 -14301.705} C_VEL
LIN {X 0,Y 341.029,Z 532.816,A -85,B 0,C 180,E1 -14304.086,E2 -14304.086} C_VEL
LIN {X 0,Y 341.172,Z 532.802,A -85,B 0,C 180,E1 -14307.639,E2 -14307.639} C_VEL
LIN {X 0,Y 341.3,Z 532.784,A -85,B 0,C 180,E1 -14310,E2 -14310} C_VEL
LIN {X 0,Y 341.172,Z 532.797,A -85,B 0,C 180,E1 -14312.361,E2 -14312.361} C_VEL
LIN {X 0,Y 341.02,Z 532.815,A -85,B 0,C 180,E1 -14317.103,E2 -14317.103} C_VEL
LIN {X 0,Y 340.853,Z 532.836,A -85,B 0,C 180,E1 -14320.694,E2 -14320.694} C_VEL
LIN {X 0,Y 340.867,Z 532.836,A -85,B 0,C 180,E1 -14324.324,E2 -14324.324} C_VEL
LIN {X 0,Y 340.841,Z 532.838,A -85,B 0,C 180,E1 -14328.466,E2 -14328.466} C_VEL
LIN {X 0,Y 340.72,Z 532.858,A -85,B 0,C 180,E1 -14331.841,E2 -14331.841} C_VEL
LIN {X 0,Y 340.774,Z 532.849,A -85,B 0,C 180,E1 -14335.664,E2 -14335.664} C_VEL
LIN {X 0,Y 340.73,Z 532.854,A -85,B 0,C 180,E1 -14338.32,E2 -14338.32} C_VEL
LIN {X 0,Y 340.699,Z 532.855,A -85,B 0,C 180,E1 -14341.044,E2 -14341.044} C_VEL
LIN {X 0,Y 340.719,Z 532.853,A -85,B 0,C 180,E1 -14345.278,E2 -14345.278} C_VEL
LIN {X 0,Y 340.718,Z 532.855,A -85,B 0,C 180,E1 -14348.387,E2 -14348.387} C_VEL
LIN {X 0,Y 340.726,Z 532.852,A -85,B 0,C 180,E1 -14351.302,E2 -14351.302} C_VEL
LIN {X 0,Y 340.736,Z 532.852,A -85,B 0,C 180,E1 -14354.529,E2 -14354.529} C_VEL
LIN {X 0,Y 340.675,Z 532.863,A -85,B 0,C 180,E1 -14356.232,E2 -14356.232} C_VEL
LIN {X 0,Y 339.992,Z 532.944,A -85,B 0,C 180,E1 -14357.219,E2 -14357.219} C_VEL
LIN {X 0,Y 337.159,Z 533.297,A -85,B 0,C 180,E1 -14358.824,E2 -14358.824} C_VEL
LIN {X 0,Y 334.764,Z 533.6,A -85,B 0,C 180,E1 -14360.124,E2 -14360.124} C_VEL
LIN {X 0,Y 333.728,Z 533.724,A -85,B 0,C 180,E1 -14361.13,E2 -14361.13} C_VEL
LIN {X 0,Y 333.638,Z 533.734,A -85,B 0,C 180,E1 -14361.47,E2 -14361.47} C_VEL
LIN {X 0,Y 333.671,Z 533.731,A -85,B 0,C 180,E1 -14365.34,E2 -14365.34} C_VEL
LIN {X 0,Y 333.697,Z 533.728,A -85,B 0,C 180,E1 -14369.637,E2 -14369.637} C_VEL
LIN {X 0,Y 333.741,Z 533.726,A -85,B 0,C 180,E1 -14372.4,E2 -14372.4} C_VEL
LIN {X 0,Y 333.722,Z 533.724,A -85,B 0,C 180,E1 -14375.09,E2 -14375.09} C_VEL
LIN {X 0,Y 333.688,Z 533.729,A -85,B 0,C 180,E1 -14379.019,E2 -14379.019} C_VEL
LIN {X 0,Y 333.79,Z 533.716,A -85,B 0,C 180,E1 -14381.589,E2 -14381.589} C_VEL
LIN {X 0,Y 333.803,Z 533.714,A -85,B 0,C 180,E1 -14385.576,E2 -14385.576} C_VEL
LIN {X 0,Y 333.831,Z 533.711,A -85,B 0,C 180,E1 -14389.077,E2 -14389.077} C_VEL
LIN {X 0,Y 334.019,Z 533.69,A -85,B 0,C 180,E1 -14392.747,E2 -14392.747} C_VEL
LIN {X 0,Y 333.806,Z 533.714,A -85,B 0,C 180,E1 -14395.169,E2 -14395.169} C_VEL
LIN {X 0,Y 334.101,Z 533.677,A -85,B 0,C 180,E1 -14397.588,E2 -14397.588} C_VEL
LIN {X 0,Y 334.24,Z 533.661,A -85,B 0,C 180,E1 -14400,E2 -14400} C_VEL
LIN {X 0,Y 334.1,Z 533.682,A -85,B 0,C 180,E1 -14402.411,E2 -14402.411} C_VEL
LIN {X 0,Y 334.008,Z 533.69,A -85,B 0,C 180,E1 -14406.039,E2 -14406.039} C_VEL
LIN {X 0,Y 333.978,Z 533.698,A -85,B 0,C 180,E1 -14408.501,E2 -14408.501} C_VEL
LIN {X 0,Y 333.784,Z 533.718,A -85,B 0,C 180,E1 -14412.155,E2 -14412.155} C_VEL
LIN {X 0,Y 333.771,Z 533.718,A -85,B 0,C 180,E1 -14415.886,E2 -14415.886} C_VEL
LIN {X 0,Y 333.79,Z 533.722,A -85,B 0,C 180,E1 -14418.655,E2 -14418.655} C_VEL
LIN {X 0,Y 333.65,Z 533.735,A -85,B 0,C 180,E1 -14422.281,E2 -14422.281} C_VEL
LIN {X 0,Y 333.729,Z 533.725,A -85,B 0,C 180,E1 -14426.246,E2 -14426.246} C_VEL
LIN {X 0,Y 333.705,Z 533.73,A -85,B 0,C 180,E1 -14428.972,E2 -14428.972} C_VEL
LIN {X 0,Y 333.637,Z 533.739,A -85,B 0,C 180,E1 -14432.587,E2 -14432.587} C_VEL
LIN {X 0,Y 333.67,Z 533.731,A -85,B 0,C 180,E1 -14436.139,E2 -14436.139} C_VEL
LIN {X 0,Y 333.641,Z 533.737,A -85,B 0,C 180,E1 -14439.193,E2 -14439.193} C_VEL
LIN {X 0,Y 333.628,Z 533.739,A -85,B 0,C 180,E1 -14442.5,E2 -14442.5} C_VEL
LIN {X 0,Y 333.617,Z 533.737,A -85,B 0,C 180,E1 -14445.96,E2 -14445.96} C_VEL
LIN {X 0,Y 333.643,Z 533.736,A -85,B 0,C 180,E1 -14449.316,E2 -14449.316} C_VEL
LIN {X 0,Y 333.662,Z 533.736,A -85,B 0,C 180,E1 -14453.168,E2 -14453.168} C_VEL
LIN {X 0,Y 333.784,Z 533.816,A -85,B 0,C 180,E1 -14454.948,E2 -14454.948} C_VEL
LIN {X 0,Y 336.404,Z 547.445,A -85,B 0,C 180,E1 -14458.931,E2 -14458.931} C_VEL
LIN {X 0,Y 337.377,Z 553.524,A -85,B 0,C 180,E1 -14460.617,E2 -14460.617} C_VEL
LIN {X 0,Y 335.935,Z 566.842,A -85,B 0,C 180,E1 -14464.104,E2 -14464.104} C_VEL
LIN {X 0,Y 334.257,Z 584.713,A -85,B 0,C 180,E1 -14468.735,E2 -14468.735} C_VEL
LIN {X 0,Y 333.623,Z 594.492,A -85,B 0,C 180,E1 -14471.212,E2 -14471.212} C_VEL
LIN {X 0,Y 333.918,Z 600.246,A -85,B 0,C 180,E1 -14471.446,E2 -14471.446} C_VEL
LIN {X 0,Y 337.734,Z 649.541,A -85,B 0,C 180,E1 -14473.024,E2 -14473.024} C_VEL
LIN {X 0,Y 337.011,Z 680.016,A -85,B 0,C 180,E1 -14473.932,E2 -14473.932} C_VEL
LIN {X 0,Y 336.476,Z 692.399,A -85,B 0,C 180,E1 -14474.555,E2 -14474.555} C_VEL
LIN {X 0,Y 335.582,Z 702.823,A -85,B 0,C 180,E1 -14475.29,E2 -14475.29} C_VEL
LIN {X 0,Y 334.961,Z 712.521,A -85,B 0,C 180,E1 -14476.192,E2 -14476.192} C_VEL
LIN {X 0,Y 334.127,Z 722.703,A -85,B 0,C 180,E1 -14477.395,E2 -14477.395} C_VEL
LIN {X 0,Y 333.373,Z 731.719,A -85,B 0,C 180,E1 -14478.755,E2 -14478.755} C_VEL
LIN {X 0,Y 332.962,Z 739.784,A -85,B 0,C 180,E1 -14480.279,E2 -14480.279} C_VEL
LIN {X 0,Y 332.786,Z 747.334,A -85,B 0,C 180,E1 -14482.11,E2 -14482.11} C_VEL
LIN {X 0,Y 332.83,Z 753.011,A -85,B 0,C 180,E1 -14483.94,E2 -14483.94} C_VEL
LIN {X 0,Y 333.068,Z 757.171,A -85,B 0,C 180,E1 -14485.765,E2 -14485.765} C_VEL
LIN {X 0,Y 333.219,Z 759.869,A -85,B 0,C 180,E1 -14487.582,E2 -14487.582} C_VEL
LIN {X 0,Y 333.392,Z 760.981,A -85,B 0,C 180,E1 -14488.792,E2 -14488.792} C_VEL
LIN {X 0,Y 333.633,Z 761.506,A -85,B 0,C 180,E1 -14490,E2 -14490} C_VEL
LIN {X 0,Y 333.254,Z 761.423,A -85,B 0,C 180,E1 -14491.208,E2 -14491.208} C_VEL
LIN {X 0,Y 333.109,Z 760.802,A -85,B 0,C 180,E1 -14492.418,E2 -14492.418} C_VEL
LIN {X 0,Y 333.021,Z 759.668,A -85,B 0,C 180,E1 -14493.63,E2 -14493.63} C_VEL
LIN {X 0,Y 332.682,Z 756.885,A -85,B 0,C 180,E1 -14495.455,E2 -14495.455} C_VEL
LIN {X 0,Y 332.566,Z 752.837,A -85,B 0,C 180,E1 -14497.284,E2 -14497.284} C_VEL
LIN {X 0,Y 332.723,Z 747.349,A -85,B 0,C 180,E1 -14499.115,E2 -14499.115} C_VEL
LIN {X 0,Y 333.175,Z 740.285,A -85,B 0,C 180,E1 -14500.943,E2 -14500.943} C_VEL
LIN {X 0,Y 333.957,Z 732.897,A -85,B 0,C 180,E1 -14502.457,E2 -14502.457} C_VEL
LIN {X 0,Y 335.15,Z 723.817,A -85,B 0,C 180,E1 -14503.954,E2 -14503.954} C_VEL
LIN {X 0,Y 336.411,Z 713.565,A -85,B 0,C 180,E1 -14505.292,E2 -14505.292} C_VEL
LIN {X 0,Y 337.737,Z 703.619,A -85,B 0,C 180,E1 -14506.315,E2 -14506.315} C_VEL
LIN {X 0,Y 339.044,Z 691.827,A -85,B 0,C 180,E1 -14507.258,E2 -14507.258} C_VEL
LIN {X 0,Y 340.203,Z 678.956,A -85,B 0,C 180,E1 -14507.999,E2 -14507.999} C_VEL
LIN {X 0,Y 340.981,Z 665.485,A -85,B 0,C 180,E1 -14508.513,E2 -14508.513} C_VEL
LIN {X 0,Y 341.356,Z 648.357,A -85,B 0,C 180,E1 -14508.998,E2 -14508.998} C_VEL
LIN {X 0,Y 340.035,Z 621.732,A -85,B 0,C 180,E1 -14509.917,E2 -14509.917} C_VEL
LIN {X 0,Y 337.889,Z 602.475,A -85,B 0,C 180,E1 -14510.707,E2 -14510.707} C_VEL
LIN {X 0,Y 334.575,Z 583.086,A -85,B 0,C 180,E1 -14511.653,E2 -14511.653} C_VEL
LIN {X 0,Y 334.189,Z 580.25,A -85,B 0,C 180,E1 -14511.836,E2 -14511.836} C_VEL
LIN {X 0,Y 335.113,Z 568.644,A -85,B 0,C 180,E1 -14514.799,E2 -14514.799} C_VEL
LIN {X 0,Y 336.873,Z 552.993,A -85,B 0,C 180,E1 -14519.014,E2 -14519.014} C_VEL
LIN {X 0,Y 336.788,Z 549.387,A -85,B 0,C 180,E1 -14520.054,E2 -14520.054} C_VEL
LIN {X 0,Y 334.986,Z 539.858,A -85,B 0,C 180,E1 -14523.056,E2 -14523.056} C_VEL
LIN {X 0,Y 333.722,Z 533.775,A -85,B 0,C 180,E1 -14525.175,E2 -14525.175} C_VEL
LIN {X 0,Y 333.642,Z 533.74,A -85,B 0,C 180,E1 -14529.192,E2 -14529.192} C_VEL
LIN {X 0,Y 333.629,Z 533.736,A -85,B 0,C 180,E1 -14532.5,E2 -14532.5} C_VEL
LIN {X 0,Y 333.664,Z 533.734,A -85,B 0,C 180,E1 -14535.967,E2 -14535.967} C_VEL
LIN {X 0,Y 333.696,Z 533.732,A -85,B 0,C 180,E1 -14539.304,E2 -14539.304} C_VEL
LIN {X 0,Y 333.662,Z 533.733,A -85,B 0,C 180,E1 -14543.167,E2 -14543.167} C_VEL
LIN {X 0,Y 333.635,Z 533.735,A -85,B 0,C 180,E1 -14546.792,E2 -14546.792} C_VEL
LIN {X 0,Y 333.698,Z 533.728,A -85,B 0,C 180,E1 -14549.709,E2 -14549.709} C_VEL
LIN {X 0,Y 333.737,Z 533.727,A -85,B 0,C 180,E1 -14552.401,E2 -14552.401} C_VEL
LIN {X 0,Y 333.719,Z 533.73,A -85,B 0,C 180,E1 -14555.091,E2 -14555.091} C_VEL
LIN {X 0,Y 333.672,Z 533.731,A -85,B 0,C 180,E1 -14559.019,E2 -14559.019} C_VEL
LIN {X 0,Y 333.786,Z 533.717,A -85,B 0,C 180,E1 -14561.589,E2 -14561.589} C_VEL
LIN {X 0,Y 333.8,Z 533.719,A -85,B 0,C 180,E1 -14565.577,E2 -14565.577} C_VEL
LIN {X 0,Y 333.83,Z 533.713,A -85,B 0,C 180,E1 -14569.078,E2 -14569.078} C_VEL
LIN {X 0,Y 334.02,Z 533.691,A -85,B 0,C 180,E1 -14572.748,E2 -14572.748} C_VEL
LIN {X 0,Y 333.81,Z 533.719,A -85,B 0,C 180,E1 -14575.17,E2 -14575.17} C_VEL
LIN {X 0,Y 334.156,Z 533.912,A -85,B 0,C 180,E1 -14577.691,E2 -14577.691} C_VEL
LIN {X 0,Y 334.386,Z 534.988,A -85,B 0,C 180,E1 -14577.896,E2 -14577.896} C_VEL
LIN {X 0,Y 340.538,Z 546.895,A -85,B 0,C 180,E1 -14578.86,E2 -14578.86} C_VEL
LIN {X 0,Y 344.509,Z 555.956,A -85,B 0,C 180,E1 -14579.469,E2 -14579.469} C_VEL
LIN {X 0,Y 344.447,Z 576.703,A -85,B 0,C 180,E1 -14580.062,E2 -14580.062} C_VEL
LIN {X 0,Y 344.295,Z 587.867,A -85,B 0,C 180,E1 -14580.593,E2 -14580.593} C_VEL
LIN {X 0,Y 343.825,Z 598.998,A -85,B 0,C 180,E1 -14581.318,E2 -14581.318} C_VEL
LIN {X 0,Y 342.967,Z 610.929,A -85,B 0,C 180,E1 -14582.349,E2 -14582.349} C_VEL
LIN {X 0,Y 342.017,Z 621.539,A -85,B 0,C 180,E1 -14583.535,E2 -14583.535} C_VEL
LIN {X 0,Y 341.049,Z 630.11,A -85,B 0,C 180,E1 -14584.729,E2 -14584.729} C_VEL
LIN {X 0,Y 339.888,Z 638.921,A -85,B 0,C 180,E1 -14586.244,E2 -14586.244} C_VEL
LIN {X 0,Y 338.817,Z 646.029,A -85,B 0,C 180,E1 -14587.749,E2 -14587.749} C_VEL
LIN {X 0,Y 337.625,Z 652.976,A -85,B 0,C 180,E1 -14589.586,E2 -14589.586} C_VEL
LIN {X 0,Y 336.609,Z 658.539,A -85,B 0,C 180,E1 -14591.511,E2 -14591.511} C_VEL
LIN {X 0,Y 335.76,Z 662.505,A -85,B 0,C 180,E1 -14593.312,E2 -14593.312} C_VEL
LIN {X 0,Y 335.039,Z 665.499,A -85,B 0,C 180,E1 -14595.225,E2 -14595.225} C_VEL
LIN {X 0,Y 334.529,Z 667.31,A -85,B 0,C 180,E1 -14597.105,E2 -14597.105} C_VEL
LIN {X 0,Y 334.177,Z 668.04,A -85,B 0,C 180,E1 -14598.851,E2 -14598.851} C_VEL
LIN {X 0,Y 333.95,Z 667.744,A -85,B 0,C 180,E1 -14600.964,E2 -14600.964} C_VEL
LIN {X 0,Y 333.848,Z 666.906,A -85,B 0,C 180,E1 -14602.268,E2 -14602.268} C_VEL
LIN {X 0,Y 333.87,Z 665.596,A -85,B 0,C 180,E1 -14603.576,E2 -14603.576} C_VEL
LIN {X 0,Y 334.017,Z 663.196,A -85,B 0,C 180,E1 -14605.213,E2 -14605.213} C_VEL
LIN {X 0,Y 334.258,Z 659.891,A -85,B 0,C 180,E1 -14606.876,E2 -14606.876} C_VEL
LIN {X 0,Y 334.635,Z 654.63,A -85,B 0,C 180,E1 -14608.885,E2 -14608.885} C_VEL
LIN {X 0,Y 335.143,Z 648.432,A -85,B 0,C 180,E1 -14610.711,E2 -14610.711} C_VEL
LIN {X 0,Y 335.805,Z 640.339,A -85,B 0,C 180,E1 -14612.611,E2 -14612.611} C_VEL
LIN {X 0,Y 336.56,Z 631.109,A -85,B 0,C 180,E1 -14614.32,E2 -14614.32} C_VEL
LIN {X 0,Y 337.382,Z 620.728,A -85,B 0,C 180,E1 -14615.865,E2 -14615.865} C_VEL
LIN {X 0,Y 338.057,Z 609.151,A -85,B 0,C 180,E1 -14617.225,E2 -14617.225} C_VEL
LIN {X 0,Y 338.71,Z 597.558,A -85,B 0,C 180,E1 -14618.292,E2 -14618.292} C_VEL
LIN {X 0,Y 339.12,Z 584.348,A -85,B 0,C 180,E1 -14619.205,E2 -14619.205} C_VEL
LIN {X 0,Y 339.34,Z 571.999,A -85,B 0,C 180,E1 -14619.812,E2 -14619.812} C_VEL
LIN {X 0,Y 339.394,Z 555.949,A -85,B 0,C 180,E1 -14620.288,E2 -14620.288} C_VEL
LIN {X 0,Y 339.226,Z 551.052,A -85,B 0,C 180,E1 -14620.416,E2 -14620.416} C_VEL
LIN {X 0,Y 333.822,Z 534.533,A -85,B 0,C 180,E1 -14621.098,E2 -14621.098} C_VEL
LIN {X 0,Y 333.69,Z 533.793,A -85,B 0,C 180,E1 -14621.334,E2 -14621.334} C_VEL
LIN {X 0,Y 333.678,Z 533.732,A -85,B 0,C 180,E1 -14625.736,E2 -14625.736} C_VEL
LIN {X 0,Y 333.701,Z 533.732,A -85,B 0,C 180,E1 -14629.306,E2 -14629.306} C_VEL
LIN {X 0,Y 333.666,Z 533.734,A -85,B 0,C 180,E1 -14633.169,E2 -14633.169} C_VEL
LIN {X 0,Y 333.674,Z 533.735,A -85,B 0,C 180,E1 -14635.342,E2 -14635.342} C_VEL
LIN {X 0,Y 333.704,Z 533.73,A -85,B 0,C 180,E1 -14639.711,E2 -14639.711} C_VEL
LIN {X 0,Y 333.745,Z 533.721,A -85,B 0,C 180,E1 -14642.402,E2 -14642.402} C_VEL
LIN {X 0,Y 333.729,Z 533.725,A -85,B 0,C 180,E1 -14645.092,E2 -14645.092} C_VEL
LIN {X 0,Y 333.68,Z 533.731,A -85,B 0,C 180,E1 -14649.02,E2 -14649.02} C_VEL
LIN {X 0,Y 333.744,Z 533.728,A -85,B 0,C 180,E1 -14651.587,E2 -14651.587} C_VEL
LIN {X 0,Y 333.812,Z 533.719,A -85,B 0,C 180,E1 -14655.577,E2 -14655.577} C_VEL
LIN {X 0,Y 333.838,Z 533.711,A -85,B 0,C 180,E1 -14659.079,E2 -14659.079} C_VEL
LIN {X 0,Y 333.973,Z 533.693,A -85,B 0,C 180,E1 -14662.747,E2 -14662.747} C_VEL
LIN {X 0,Y 333.806,Z 533.715,A -85,B 0,C 180,E1 -14665.169,E2 -14665.169} C_VEL
LIN {X 0,Y 334.109,Z 533.681,A -85,B 0,C 180,E1 -14667.589,E2 -14667.589} C_VEL
LIN {X 0,Y 334.25,Z 533.662,A -85,B 0,C 180,E1 -14670,E2 -14670} C_VEL
LIN {X 0,Y 334.109,Z 533.677,A -85,B 0,C 180,E1 -14672.411,E2 -14672.411} C_VEL
LIN {X 0,Y 334.003,Z 533.693,A -85,B 0,C 180,E1 -14676.039,E2 -14676.039} C_VEL
LIN {X 0,Y 333.825,Z 533.716,A -85,B 0,C 180,E1 -14679.696,E2 -14679.696} C_VEL
LIN {X 0,Y 333.801,Z 533.716,A -85,B 0,C 180,E1 -14683.391,E2 -14683.391} C_VEL
LIN {X 0,Y 333.75,Z 533.721,A -85,B 0,C 180,E1 -14687.146,E2 -14687.146} C_VEL
LIN {X 0,Y 333.738,Z 533.726,A -85,B 0,C 180,E1 -14689.69,E2 -14689.69} C_VEL
LIN {X 0,Y 333.672,Z 533.733,A -85,B 0,C 180,E1 -14693.59,E2 -14693.59} C_VEL
LIN {X 0,Y 333.737,Z 533.725,A -85,B 0,C 180,E1 -14696.246,E2 -14696.246} C_VEL
LIN {X 0,Y 333.692,Z 533.728,A -85,B 0,C 180,E1 -14698.973,E2 -14698.973} C_VEL
LIN {X 0,Y 333.647,Z 533.734,A -85,B 0,C 180,E1 -14702.587,E2 -14702.587} C_VEL
LIN {X 0,Y 333.677,Z 533.735,A -85,B 0,C 180,E1 -14706.138,E2 -14706.138} C_VEL
LIN {X 0,Y 333.684,Z 533.729,A -85,B 0,C 180,E1 -14709.186,E2 -14709.186} C_VEL
LIN {X 0,Y 333.691,Z 533.73,A -85,B 0,C 180,E1 -14712.51,E2 -14712.51} C_VEL
LIN {X 0,Y 333.634,Z 533.74,A -85,B 0,C 180,E1 -14715.96,E2 -14715.96} C_VEL
LIN {X 0,Y 333.645,Z 533.734,A -85,B 0,C 180,E1 -14719.314,E2 -14719.314} C_VEL
LIN {X 0,Y 333.638,Z 533.734,A -85,B 0,C 180,E1 -14721.47,E2 -14721.47} C_VEL
LIN {X 0,Y 332.951,Z 533.824,A -85,B 0,C 180,E1 -14722.479,E2 -14722.479} C_VEL
LIN {X 0,Y 330.08,Z 534.183,A -85,B 0,C 180,E1 -14724.119,E2 -14724.119} C_VEL
LIN {X 0,Y 327.677,Z 534.479,A -85,B 0,C 180,E1 -14725.448,E2 -14725.448} C_VEL
LIN {X 0,Y 326.675,Z 534.605,A -85,B 0,C 180,E1 -14726.476,E2 -14726.476} C_VEL
LIN {X 0,Y 326.607,Z 534.61,A -85,B 0,C 180,E1 -14726.825,E2 -14726.825} C_VEL
LIN {X 0,Y 326.658,Z 534.609,A -85,B 0,C 180,E1 -14730.34,E2 -14730.34} C_VEL
LIN {X 0,Y 326.686,Z 534.604,A -85,B 0,C 180,E1 -14734.515,E2 -14734.515} C_VEL
LIN {X 0,Y 326.648,Z 534.609,A -85,B 0,C 180,E1 -14738.545,E2 -14738.545} C_VEL
LIN {X 0,Y 326.74,Z 534.594,A -85,B 0,C 180,E1 -14741.177,E2 -14741.177} C_VEL
LIN {X 0,Y 326.758,Z 534.592,A -85,B 0,C 180,E1 -14745.432,E2 -14745.432} C_VEL
LIN {X 0,Y 326.767,Z 534.592,A -85,B 0,C 180,E1 -14748.838,E2 -14748.838} C_VEL
LIN {X 0,Y 326.973,Z 534.569,A -85,B 0,C 180,E1 -14752.59,E2 -14752.59} C_VEL
LIN {X 0,Y 326.773,Z 534.591,A -85,B 0,C 180,E1 -14755.064,E2 -14755.064} C_VEL
LIN {X 0,Y 327.042,Z 534.556,A -85,B 0,C 180,E1 -14757.536,E2 -14757.536} C_VEL
LIN {X 0,Y 327.191,Z 534.539,A -85,B 0,C 180,E1 -14760,E2 -14760} C_VEL
LIN {X 0,Y 327.041,Z 534.562,A -85,B 0,C 180,E1 -14762.463,E2 -14762.463} C_VEL
LIN {X 0,Y 326.983,Z 534.566,A -85,B 0,C 180,E1 -14766.169,E2 -14766.169} C_VEL
LIN {X 0,Y 326.908,Z 534.578,A -85,B 0,C 180,E1 -14768.655,E2 -14768.655} C_VEL
LIN {X 0,Y 326.727,Z 534.6,A -85,B 0,C 180,E1 -14772.421,E2 -14772.421} C_VEL
LIN {X 0,Y 326.747,Z 534.596,A -85,B 0,C 180,E1 -14774.957,E2 -14774.957} C_VEL
LIN {X 0,Y 326.726,Z 534.6,A -85,B 0,C 180,E1 -14778.838,E2 -14778.838} C_VEL
LIN {X 0,Y 326.596,Z 534.617,A -85,B 0,C 180,E1 -14782.789,E2 -14782.789} C_VEL
LIN {X 0,Y 326.683,Z 534.601,A -85,B 0,C 180,E1 -14785.484,E2 -14785.484} C_VEL
LIN {X 0,Y 326.655,Z 534.604,A -85,B 0,C 180,E1 -14789.659,E2 -14789.659} C_VEL
LIN {X 0,Y 326.601,Z 534.612,A -85,B 0,C 180,E1 -14794.02,E2 -14794.02} C_VEL
LIN {X 0,Y 326.622,Z 534.61,A -85,B 0,C 180,E1 -14797.239,E2 -14797.239} C_VEL
LIN {X 0,Y 326.572,Z 534.618,A -85,B 0,C 180,E1 -14801.132,E2 -14801.132} C_VEL
LIN {X 0,Y 326.552,Z 534.622,A -85,B 0,C 180,E1 -14804.748,E2 -14804.748} C_VEL
LIN {X 0,Y 326.572,Z 534.615,A -85,B 0,C 180,E1 -14808.155,E2 -14808.155} C_VEL
LIN {X 0,Y 326.62,Z 534.61,A -85,B 0,C 180,E1 -14811.392,E2 -14811.392} C_VEL
LIN {X 0,Y 326.76,Z 534.771,A -85,B 0,C 180,E1 -14814.816,E2 -14814.816} C_VEL
LIN {X 0,Y 329.623,Z 549.656,A -85,B 0,C 180,E1 -14819.223,E2 -14819.223} C_VEL
LIN {X 0,Y 330.334,Z 553.633,A -85,B 0,C 180,E1 -14820.354,E2 -14820.354} C_VEL
LIN {X 0,Y 328.969,Z 566.464,A -85,B 0,C 180,E1 -14823.802,E2 -14823.802} C_VEL
LIN {X 0,Y 327.201,Z 584.438,A -85,B 0,C 180,E1 -14828.584,E2 -14828.584} C_VEL
LIN {X 0,Y 326.604,Z 593.217,A -85,B 0,C 180,E1 -14830.876,E2 -14830.876} C_VEL
LIN {X 0,Y 326.934,Z 599.141,A -85,B 0,C 180,E1 -14831.123,E2 -14831.123} C_VEL
LIN {X 0,Y 330.757,Z 650.586,A -85,B 0,C 180,E1 -14832.82,E2 -14832.82} C_VEL
LIN {X 0,Y 330.09,Z 678.379,A -85,B 0,C 180,E1 -14833.671,E2 -14833.671} C_VEL
LIN {X 0,Y 329.549,Z 690.849,A -85,B 0,C 180,E1 -14834.302,E2 -14834.302} C_VEL
LIN {X 0,Y 328.559,Z 702.275,A -85,B 0,C 180,E1 -14835.127,E2 -14835.127} C_VEL
LIN {X 0,Y 327.917,Z 711.842,A -85,B 0,C 180,E1 -14836.048,E2 -14836.048} C_VEL
LIN {X 0,Y 327.112,Z 721.954,A -85,B 0,C 180,E1 -14837.278,E2 -14837.278} C_VEL
LIN {X 0,Y 326.27,Z 731.805,A -85,B 0,C 180,E1 -14838.822,E2 -14838.822} C_VEL
LIN {X 0,Y 325.894,Z 739.613,A -85,B 0,C 180,E1 -14840.379,E2 -14840.379} C_VEL
LIN {X 0,Y 325.716,Z 745.864,A -85,B 0,C 180,E1 -14841.938,E2 -14841.938} C_VEL
LIN {X 0,Y 325.784,Z 751.666,A -85,B 0,C 180,E1 -14843.808,E2 -14843.808} C_VEL
LIN {X 0,Y 326.023,Z 755.917,A -85,B 0,C 180,E1 -14845.673,E2 -14845.673} C_VEL
LIN {X 0,Y 326.187,Z 758.697,A -85,B 0,C 180,E1 -14847.53,E2 -14847.53} C_VEL
LIN {X 0,Y 326.381,Z 759.854,A -85,B 0,C 180,E1 -14848.766,E2 -14848.766} C_VEL
LIN {X 0,Y 326.619,Z 760.432,A -85,B 0,C 180,E1 -14850,E2 -14850} C_VEL
LIN {X 0,Y 326.217,Z 760.391,A -85,B 0,C 180,E1 -14851.234,E2 -14851.234} C_VEL
LIN {X 0,Y 326.059,Z 759.809,A -85,B 0,C 180,E1 -14852.471,E2 -14852.471} C_VEL
LIN {X 0,Y 325.932,Z 758.721,A -85,B 0,C 180,E1 -14853.709,E2 -14853.709} C_VEL
LIN {X 0,Y 325.602,Z 755.994,A -85,B 0,C 180,E1 -14855.574,E2 -14855.574} C_VEL
LIN {X 0,Y 325.481,Z 752.009,A -85,B 0,C 180,E1 -14857.444,E2 -14857.444} C_VEL
LIN {X 0,Y 325.65,Z 746.653,A -85,B 0,C 180,E1 -14859.315,E2 -14859.315} C_VEL
LIN {X 0,Y 326.144,Z 739.705,A -85,B 0,C 180,E1 -14861.182,E2 -14861.182} C_VEL
LIN {X 0,Y 327.021,Z 732.462,A -85,B 0,C 180,E1 -14862.725,E2 -14862.725} C_VEL
LIN {X 0,Y 328.268,Z 723.523,A -85,B 0,C 180,E1 -14864.253,E2 -14864.253} C_VEL
LIN {X 0,Y 329.57,Z 713.488,A -85,B 0,C 180,E1 -14865.618,E2 -14865.618} C_VEL
LIN {X 0,Y 331.171,Z 702.353,A -85,B 0,C 180,E1 -14866.806,E2 -14866.806} C_VEL
LIN {X 0,Y 332.494,Z 691.001,A -85,B 0,C 180,E1 -14867.741,E2 -14867.741} C_VEL
LIN {X 0,Y 333.679,Z 678.578,A -85,B 0,C 180,E1 -14868.491,E2 -14868.491} C_VEL
LIN {X 0,Y 334.533,Z 666.114,A -85,B 0,C 180,E1 -14869.003,E2 -14869.003} C_VEL
LIN {X 0,Y 334.955,Z 648.948,A -85,B 0,C 180,E1 -14869.505,E2 -14869.505} C_VEL
LIN {X 0,Y 333.675,Z 621.852,A -85,B 0,C 180,E1 -14870.468,E2 -14870.468} C_VEL
LIN {X 0,Y 331.46,Z 602.52,A -85,B 0,C 180,E1 -14871.311,E2 -14871.311} C_VEL
LIN {X 0,Y 328.004,Z 582.313,A -85,B 0,C 180,E1 -14872.335,E2 -14872.335} C_VEL
LIN {X 0,Y 327.356,Z 578.277,A -85,B 0,C 180,E1 -14872.607,E2 -14872.607} C_VEL
LIN {X 0,Y 328.781,Z 563.023,A -85,B 0,C 180,E1 -14876.672,E2 -14876.672} C_VEL
LIN {X 0,Y 329.959,Z 553.53,A -85,B 0,C 180,E1 -14879.333,E2 -14879.333} C_VEL
LIN {X 0,Y 329.704,Z 549.921,A -85,B 0,C 180,E1 -14880.414,E2 -14880.414} C_VEL
LIN {X 0,Y 327.689,Z 539.3,A -85,B 0,C 180,E1 -14883.891,E2 -14883.891} C_VEL
LIN {X 0,Y 326.658,Z 534.632,A -85,B 0,C 180,E1 -14885.631,E2 -14885.631} C_VEL
LIN {X 0,Y 326.607,Z 534.616,A -85,B 0,C 180,E1 -14889.227,E2 -14889.227} C_VEL
LIN {X 0,Y 326.581,Z 534.617,A -85,B 0,C 180,E1 -14892.973,E2 -14892.973} C_VEL
LIN {X 0,Y 326.622,Z 534.609,A -85,B 0,C 180,E1 -14897.018,E2 -14897.018} C_VEL
LIN {X 0,Y 326.642,Z 534.604,A -85,B 0,C 180,E1 -14900.765,E2 -14900.765} C_VEL
LIN {X 0,Y 326.607,Z 534.607,A -85,B 0,C 180,E1 -14904.48,E2 -14904.48} C_VEL
LIN {X 0,Y 326.608,Z 534.607,A -85,B 0,C 180,E1 -14907.456,E2 -14907.456} C_VEL
LIN {X 0,Y 326.655,Z 534.603,A -85,B 0,C 180,E1 -14910.341,E2 -14910.341} C_VEL
LIN {X 0,Y 326.683,Z 534.6,A -85,B 0,C 180,E1 -14914.516,E2 -14914.516} C_VEL
LIN {X 0,Y 326.638,Z 534.611,A -85,B 0,C 180,E1 -14918.545,E2 -14918.545} C_VEL
LIN {X 0,Y 326.737,Z 534.598,A -85,B 0,C 180,E1 -14921.177,E2 -14921.177} C_VEL
LIN {X 0,Y 326.755,Z 534.595,A -85,B 0,C 180,E1 -14925.433,E2 -14925.433} C_VEL
LIN {X 0,Y 326.766,Z 534.594,A -85,B 0,C 180,E1 -14928.839,E2 -14928.839} C_VEL
LIN {X 0,Y 326.973,Z 534.569,A -85,B 0,C 180,E1 -14932.591,E2 -14932.591} C_VEL
LIN {X 0,Y 326.777,Z 534.595,A -85,B 0,C 180,E1 -14935.065,E2 -14935.065} C_VEL
LIN {X 0,Y 326.924,Z 534.691,A -85,B 0,C 180,E1 -14936.843,E2 -14936.843} C_VEL
LIN {X 0,Y 327.1,Z 535.429,A -85,B 0,C 180,E1 -14937.075,E2 -14937.075} C_VEL
LIN {X 0,Y 328.649,Z 538.34,A -85,B 0,C 180,E1 -14937.385,E2 -14937.385} C_VEL
LIN {X 0,Y 335.003,Z 550.485,A -85,B 0,C 180,E1 -14938.415,E2 -14938.415} C_VEL
LIN {X 0,Y 338.245,Z 557.845,A -85,B 0,C 180,E1 -14938.94,E2 -14938.94} C_VEL
LIN {X 0,Y 338.198,Z 577.771,A -85,B 0,C 180,E1 -14939.524,E2 -14939.524} C_VEL
LIN {X 0,Y 338.037,Z 589.283,A -85,B 0,C 180,E1 -14940.082,E2 -14940.082} C_VEL
LIN {X 0,Y 337.514,Z 600.546,A -85,B 0,C 180,E1 -14940.835,E2 -14940.835} C_VEL
LIN {X 0,Y 336.536,Z 612.958,A -85,B 0,C 180,E1 -14941.945,E2 -14941.945} C_VEL
LIN {X 0,Y 335.511,Z 623.33,A -85,B 0,C 180,E1 -14943.153,E2 -14943.153} C_VEL
LIN {X 0,Y 334.383,Z 632.694,A -85,B 0,C 180,E1 -14944.521,E2 -14944.521} C_VEL
LIN {X 0,Y 333.144,Z 641.243,A -85,B 0,C 180,E1 -14946.055,E2 -14946.055} C_VEL
LIN {X 0,Y 332.004,Z 648.211,A -85,B 0,C 180,E1 -14947.603,E2 -14947.603} C_VEL
LIN {X 0,Y 330.961,Z 653.916,A -85,B 0,C 180,E1 -14949.165,E2 -14949.165} C_VEL
LIN {X 0,Y 329.743,Z 660.101,A -85,B 0,C 180,E1 -14951.363,E2 -14951.363} C_VEL
LIN {X 0,Y 328.934,Z 663.506,A -85,B 0,C 180,E1 -14952.965,E2 -14952.965} C_VEL
LIN {X 0,Y 327.999,Z 667.058,A -85,B 0,C 180,E1 -14955.38,E2 -14955.38} C_VEL
LIN {X 0,Y 327.433,Z 668.717,A -85,B 0,C 180,E1 -14957.488,E2 -14957.488} C_VEL
LIN {X 0,Y 327.127,Z 669.158,A -85,B 0,C 180,E1 -14959.044,E2 -14959.044} C_VEL
LIN {X 0,Y 326.87,Z 668.488,A -85,B 0,C 180,E1 -14961.44,E2 -14961.44} C_VEL
LIN {X 0,Y 326.816,Z 667.425,A -85,B 0,C 180,E1 -14962.774,E2 -14962.774} C_VEL
LIN {X 0,Y 326.938,Z 664.851,A -85,B 0,C 180,E1 -14964.783,E2 -14964.783} C_VEL
LIN {X 0,Y 327.222,Z 661.034,A -85,B 0,C 180,E1 -14966.811,E2 -14966.811} C_VEL
LIN {X 0,Y 327.581,Z 655.705,A -85,B 0,C 180,E1 -14968.894,E2 -14968.894} C_VEL
LIN {X 0,Y 328.164,Z 648.855,A -85,B 0,C 180,E1 -14970.93,E2 -14970.93} C_VEL
LIN {X 0,Y 328.768,Z 641.53,A -85,B 0,C 180,E1 -14972.668,E2 -14972.668} C_VEL
LIN {X 0,Y 329.561,Z 632.336,A -85,B 0,C 180,E1 -14974.411,E2 -14974.411} C_VEL
LIN {X 0,Y 330.353,Z 622.208,A -85,B 0,C 180,E1 -14975.96,E2 -14975.96} C_VEL
LIN {X 0,Y 331.009,Z 611.764,A -85,B 0,C 180,E1 -14977.238,E2 -14977.238} C_VEL
LIN {X 0,Y 331.671,Z 600.069,A -85,B 0,C 180,E1 -14978.372,E2 -14978.372} C_VEL
LIN {X 0,Y 332.153,Z 588.541,A -85,B 0,C 180,E1 -14979.235,E2 -14979.235} C_VEL
LIN {X 0,Y 332.388,Z 574.99,A -85,B 0,C 180,E1 -14979.965,E2 -14979.965} C_VEL
LIN {X 0,Y 332.464,Z 561.581,A -85,B 0,C 180,E1 -14980.422,E2 -14980.422} C_VEL
LIN {X 0,Y 332.325,Z 552.354,A -85,B 0,C 180,E1 -14980.672,E2 -14980.672} C_VEL
LIN {X 0,Y 326.798,Z 535.454,A -85,B 0,C 180,E1 -14981.38,E2 -14981.38} C_VEL
LIN {X 0,Y 326.621,Z 534.668,A -85,B 0,C 180,E1 -14981.642,E2 -14981.642} C_VEL
LIN {X 0,Y 326.597,Z 534.617,A -85,B 0,C 180,E1 -14985.246,E2 -14985.246} C_VEL
LIN {X 0,Y 326.628,Z 534.609,A -85,B 0,C 180,E1 -14988.86,E2 -14988.86} C_VEL
LIN {X 0,Y 326.647,Z 534.611,A -85,B 0,C 180,E1 -14991.396,E2 -14991.396} C_VEL
LIN {X 0,Y 326.62,Z 534.61,A -85,B 0,C 180,E1 -14994.852,E2 -14994.852} C_VEL
LIN {X 0,Y 326.608,Z 534.616,A -85,B 0,C 180,E1 -14997.457,E2 -14997.457} C_VEL
LIN {X 0,Y 326.662,Z 534.604,A -85,B 0,C 180,E1 -15000.342,E2 -15000.342} C_VEL
LIN {X 0,Y 326.692,Z 534.6,A -85,B 0,C 180,E1 -15004.517,E2 -15004.517} C_VEL
LIN {X 0,Y 326.647,Z 534.605,A -85,B 0,C 180,E1 -15008.546,E2 -15008.546} C_VEL
LIN {X 0,Y 326.71,Z 534.6,A -85,B 0,C 180,E1 -15011.176,E2 -15011.176} C_VEL
LIN {X 0,Y 326.766,Z 534.595,A -85,B 0,C 180,E1 -15015.434,E2 -15015.434} C_VEL
LIN {X 0,Y 326.774,Z 534.59,A -85,B 0,C 180,E1 -15018.839,E2 -15018.839} C_VEL
LIN {X 0,Y 326.927,Z 534.571,A -85,B 0,C 180,E1 -15022.589,E2 -15022.589} C_VEL
LIN {X 0,Y 326.773,Z 534.591,A -85,B 0,C 180,E1 -15025.065,E2 -15025.065} C_VEL
LIN {X 0,Y 327.049,Z 534.56,A -85,B 0,C 180,E1 -15027.537,E2 -15027.537} C_VEL
LIN {X 0,Y 327.202,Z 534.54,A -85,B 0,C 180,E1 -15030,E2 -15030} C_VEL
LIN {X 0,Y 327.05,Z 534.556,A -85,B 0,C 180,E1 -15032.463,E2 -15032.463} C_VEL
LIN {X 0,Y 326.957,Z 534.569,A -85,B 0,C 180,E1 -15036.17,E2 -15036.17} C_VEL
LIN {X 0,Y 326.788,Z 534.593,A -85,B 0,C 180,E1 -15039.907,E2 -15039.907} C_VEL
LIN {X 0,Y 326.763,Z 534.595,A -85,B 0,C 180,E1 -15043.685,E2 -15043.685} C_VEL
LIN {X 0,Y 326.703,Z 534.601,A -85,B 0,C 180,E1 -15047.527,E2 -15047.527} C_VEL
LIN {X 0,Y 326.663,Z 534.607,A -85,B 0,C 180,E1 -15050.135,E2 -15050.135} C_VEL
LIN {X 0,Y 326.651,Z 534.609,A -85,B 0,C 180,E1 -15054.128,E2 -15054.128} C_VEL
LIN {X 0,Y 326.685,Z 534.601,A -85,B 0,C 180,E1 -15056.857,E2 -15056.857} C_VEL
LIN {X 0,Y 326.636,Z 534.608,A -85,B 0,C 180,E1 -15060.609,E2 -15060.609} C_VEL
LIN {X 0,Y 326.609,Z 534.616,A -85,B 0,C 180,E1 -15064.018,E2 -15064.018} C_VEL
LIN {X 0,Y 326.63,Z 534.608,A -85,B 0,C 180,E1 -15067.238,E2 -15067.238} C_VEL
LIN {X 0,Y 326.635,Z 534.612,A -85,B 0,C 180,E1 -15070.201,E2 -15070.201} C_VEL
LIN {X 0,Y 326.629,Z 534.609,A -85,B 0,C 180,E1 -15073.513,E2 -15073.513} C_VEL
LIN {X 0,Y 326.584,Z 534.613,A -85,B 0,C 180,E1 -15077.025,E2 -15077.025} C_VEL
LIN {X 0,Y 326.609,Z 534.611,A -85,B 0,C 180,E1 -15080.772,E2 -15080.772} C_VEL
LIN {X 0,Y 326.61,Z 534.613,A -85,B 0,C 180,E1 -15084.479,E2 -15084.479} C_VEL
LIN {X 0,Y 326.607,Z 534.61,A -85,B 0,C 180,E1 -15086.825,E2 -15086.825} C_VEL
LIN {X 0,Y 325.976,Z 534.694,A -85,B 0,C 180,E1 -15087.853,E2 -15087.853} C_VEL
LIN {X 0,Y 323.132,Z 535.044,A -85,B 0,C 180,E1 -15089.527,E2 -15089.527} C_VEL
LIN {X 0,Y 320.707,Z 535.346,A -85,B 0,C 180,E1 -15090.883,E2 -15090.883} C_VEL
LIN {X 0,Y 319.677,Z 535.477,A -85,B 0,C 180,E1 -15091.933,E2 -15091.933} C_VEL
LIN {X 0,Y 319.6,Z 535.485,A -85,B 0,C 180,E1 -15092.289,E2 -15092.289} C_VEL
LIN {X 0,Y 319.601,Z 535.483,A -85,B 0,C 180,E1 -15095.303,E2 -15095.303} C_VEL
LIN {X 0,Y 319.617,Z 535.481,A -85,B 0,C 180,E1 -15099.401,E2 -15099.401} C_VEL
LIN {X 0,Y 319.654,Z 535.48,A -85,B 0,C 180,E1 -15102.072,E2 -15102.072} C_VEL
LIN {X 0,Y 319.727,Z 535.47,A -85,B 0,C 180,E1 -15106.007,E2 -15106.007} C_VEL
LIN {X 0,Y 319.754,Z 535.466,A -85,B 0,C 180,E1 -15109.872,E2 -15109.872} C_VEL
LIN {X 0,Y 319.927,Z 535.449,A -85,B 0,C 180,E1 -15112.426,E2 -15112.426} C_VEL
LIN {X 0,Y 319.743,Z 535.467,A -85,B 0,C 180,E1 -15114.956,E2 -15114.956} C_VEL
LIN {X 0,Y 319.985,Z 535.435,A -85,B 0,C 180,E1 -15117.482,E2 -15117.482} C_VEL
LIN {X 0,Y 320.143,Z 535.417,A -85,B 0,C 180,E1 -15120,E2 -15120} C_VEL
LIN {X 0,Y 319.985,Z 535.441,A -85,B 0,C 180,E1 -15122.517,E2 -15122.517} C_VEL
LIN {X 0,Y 319.939,Z 535.445,A -85,B 0,C 180,E1 -15126.305,E2 -15126.305} C_VEL
LIN {X 0,Y 319.836,Z 535.457,A -85,B 0,C 180,E1 -15128.848,E2 -15128.848} C_VEL
LIN {X 0,Y 319.675,Z 535.479,A -85,B 0,C 180,E1 -15132.7,E2 -15132.7} C_VEL
LIN {X 0,Y 319.693,Z 535.472,A -85,B 0,C 180,E1 -15135.295,E2 -15135.295} C_VEL
LIN {X 0,Y 319.646,Z 535.479,A -85,B 0,C 180,E1 -15139.256,E2 -15139.256} C_VEL
LIN {X 0,Y 319.554,Z 535.49,A -85,B 0,C 180,E1 -15143.32,E2 -15143.32} C_VEL
LIN {X 0,Y 319.629,Z 535.481,A -85,B 0,C 180,E1 -15146.088,E2 -15146.088} C_VEL
LIN {X 0,Y 319.584,Z 535.489,A -85,B 0,C 180,E1 -15148.934,E2 -15148.934} C_VEL
LIN {X 0,Y 319.526,Z 535.493,A -85,B 0,C 180,E1 -15151.862,E2 -15151.862} C_VEL
LIN {X 0,Y 319.574,Z 535.487,A -85,B 0,C 180,E1 -15155.543,E2 -15155.543} C_VEL
LIN {X 0,Y 319.553,Z 535.489,A -85,B 0,C 180,E1 -15159.669,E2 -15159.669} C_VEL
LIN {X 0,Y 319.553,Z 535.49,A -85,B 0,C 180,E1 -15163.468,E2 -15163.468} C_VEL
LIN {X 0,Y 319.557,Z 535.493,A -85,B 0,C 180,E1 -15167.018,E2 -15167.018} C_VEL
LIN {X 0,Y 319.543,Z 535.492,A -85,B 0,C 180,E1 -15170.371,E2 -15170.371} C_VEL
LIN {X 0,Y 319.697,Z 535.523,A -85,B 0,C 180,E1 -15174.547,E2 -15174.547} C_VEL
LIN {X 0,Y 320.379,Z 539.525,A -85,B 0,C 180,E1 -15175.853,E2 -15175.853} C_VEL
LIN {X 0,Y 323.148,Z 553.393,A -85,B 0,C 180,E1 -15179.986,E2 -15179.986} C_VEL
LIN {X 0,Y 323.106,Z 556.662,A -85,B 0,C 180,E1 -15180.906,E2 -15180.906} C_VEL
LIN {X 0,Y 321.304,Z 571.926,A -85,B 0,C 180,E1 -15185.099,E2 -15185.099} C_VEL
LIN {X 0,Y 319.869,Z 587.766,A -85,B 0,C 180,E1 -15189.419,E2 -15189.419} C_VEL
LIN {X 0,Y 319.565,Z 592.219,A -85,B 0,C 180,E1 -15190.572,E2 -15190.572} C_VEL
LIN {X 0,Y 323.791,Z 650.747,A -85,B 0,C 180,E1 -15192.59,E2 -15192.59} C_VEL
LIN {X 0,Y 323.086,Z 678.19,A -85,B 0,C 180,E1 -15193.47,E2 -15193.47} C_VEL
LIN {X 0,Y 322.548,Z 690.307,A -85,B 0,C 180,E1 -15194.114,E2 -15194.114} C_VEL
LIN {X 0,Y 321.544,Z 701.583,A -85,B 0,C 180,E1 -15194.957,E2 -15194.957} C_VEL
LIN {X 0,Y 320.865,Z 711.062,A -85,B 0,C 180,E1 -15195.897,E2 -15195.897} C_VEL
LIN {X 0,Y 320.062,Z 721.119,A -85,B 0,C 180,E1 -15197.154,E2 -15197.154} C_VEL
LIN {X 0,Y 319.325,Z 730.045,A -85,B 0,C 180,E1 -15198.575,E2 -15198.575} C_VEL
LIN {X 0,Y 318.856,Z 738.013,A -85,B 0,C 180,E1 -15200.165,E2 -15200.165} C_VEL
LIN {X 0,Y 318.676,Z 745.5,A -85,B 0,C 180,E1 -15202.077,E2 -15202.077} C_VEL
LIN {X 0,Y 318.738,Z 750.304,A -85,B 0,C 180,E1 -15203.671,E2 -15203.671} C_VEL
LIN {X 0,Y 318.979,Z 754.636,A -85,B 0,C 180,E1 -15205.577,E2 -15205.577} C_VEL
LIN {X 0,Y 319.153,Z 757.524,A -85,B 0,C 180,E1 -15207.476,E2 -15207.476} C_VEL
LIN {X 0,Y 319.367,Z 758.716,A -85,B 0,C 180,E1 -15208.739,E2 -15208.739} C_VEL
LIN {X 0,Y 319.602,Z 759.358,A -85,B 0,C 180,E1 -15210,E2 -15210} C_VEL
LIN {X 0,Y 319.181,Z 759.343,A -85,B 0,C 180,E1 -15211.262,E2 -15211.262} C_VEL
LIN {X 0,Y 319.006,Z 758.815,A -85,B 0,C 180,E1 -15212.525,E2 -15212.525} C_VEL
LIN {X 0,Y 318.846,Z 757.757,A -85,B 0,C 180,E1 -15213.791,E2 -15213.791} C_VEL
LIN {X 0,Y 318.521,Z 755.128,A -85,B 0,C 180,E1 -15215.698,E2 -15215.698} C_VEL
LIN {X 0,Y 318.41,Z 751.224,A -85,B 0,C 180,E1 -15217.61,E2 -15217.61} C_VEL
LIN {X 0,Y 318.595,Z 745.972,A -85,B 0,C 180,E1 -15219.523,E2 -15219.523} C_VEL
LIN {X 0,Y 319.131,Z 739.115,A -85,B 0,C 180,E1 -15221.431,E2 -15221.431} C_VEL
LIN {X 0,Y 320.096,Z 732.029,A -85,B 0,C 180,E1 -15223.005,E2 -15223.005} C_VEL
LIN {X 0,Y 321.397,Z 723.298,A -85,B 0,C 180,E1 -15224.564,E2 -15224.564} C_VEL
LIN {X 0,Y 322.745,Z 713.614,A -85,B 0,C 180,E1 -15225.957,E2 -15225.957} C_VEL
LIN {X 0,Y 324.411,Z 702.801,A -85,B 0,C 180,E1 -15227.167,E2 -15227.167} C_VEL
LIN {X 0,Y 325.788,Z 691.861,A -85,B 0,C 180,E1 -15228.125,E2 -15228.125} C_VEL
LIN {X 0,Y 327.054,Z 680.342,A -85,B 0,C 180,E1 -15228.885,E2 -15228.885} C_VEL
LIN {X 0,Y 328.069,Z 666.969,A -85,B 0,C 180,E1 -15229.498,E2 -15229.498} C_VEL
LIN {X 0,Y 328.582,Z 649.311,A -85,B 0,C 180,E1 -15230.048,E2 -15230.048} C_VEL
LIN {X 0,Y 327.472,Z 623.48,A -85,B 0,C 180,E1 -15231.003,E2 -15231.003} C_VEL
LIN {X 0,Y 325.426,Z 604.727,A -85,B 0,C 180,E1 -15231.84,E2 -15231.84} C_VEL
LIN {X 0,Y 322.162,Z 584.861,A -85,B 0,C 180,E1 -15232.888,E2 -15232.888} C_VEL
LIN {X 0,Y 320.56,Z 576.534,A -85,B 0,C 180,E1 -15233.413,E2 -15233.413} C_VEL
LIN {X 0,Y 321.187,Z 569.514,A -85,B 0,C 180,E1 -15235.257,E2 -15235.257} C_VEL
LIN {X 0,Y 322.835,Z 556.084,A -85,B 0,C 180,E1 -15239.071,E2 -15239.071} C_VEL
LIN {X 0,Y 323.013,Z 552.874,A -85,B 0,C 180,E1 -15240.027,E2 -15240.027} C_VEL
LIN {X 0,Y 321.268,Z 543.418,A -85,B 0,C 180,E1 -15243.153,E2 -15243.153} C_VEL
LIN {X 0,Y 319.62,Z 535.55,A -85,B 0,C 180,E1 -15246.056,E2 -15246.056} C_VEL
LIN {X 0,Y 319.554,Z 535.492,A -85,B 0,C 180,E1 -15249.668,E2 -15249.668} C_VEL
LIN {X 0,Y 319.559,Z 535.493,A -85,B 0,C 180,E1 -15253.468,E2 -15253.468} C_VEL
LIN {X 0,Y 319.598,Z 535.484,A -85,B 0,C 180,E1 -15257.024,E2 -15257.024} C_VEL
LIN {X 0,Y 319.582,Z 535.485,A -85,B 0,C 180,E1 -15260.376,E2 -15260.376} C_VEL
LIN {X 0,Y 319.555,Z 535.487,A -85,B 0,C 180,E1 -15263.572,E2 -15263.572} C_VEL
LIN {X 0,Y 319.572,Z 535.487,A -85,B 0,C 180,E1 -15266.686,E2 -15266.686} C_VEL
LIN {X 0,Y 319.587,Z 535.487,A -85,B 0,C 180,E1 -15269.617,E2 -15269.617} C_VEL
LIN {X 0,Y 319.603,Z 535.488,A -85,B 0,C 180,E1 -15272.498,E2 -15272.498} C_VEL
LIN {X 0,Y 319.598,Z 535.488,A -85,B 0,C 180,E1 -15275.304,E2 -15275.304} C_VEL
LIN {X 0,Y 319.589,Z 535.488,A -85,B 0,C 180,E1 -15278.048,E2 -15278.048} C_VEL
LIN {X 0,Y 319.681,Z 535.479,A -85,B 0,C 180,E1 -15280.962,E2 -15280.962} C_VEL
LIN {X 0,Y 319.723,Z 535.47,A -85,B 0,C 180,E1 -15285.276,E2 -15285.276} C_VEL
LIN {X 0,Y 319.752,Z 535.47,A -85,B 0,C 180,E1 -15289.873,E2 -15289.873} C_VEL
LIN {X 0,Y 319.927,Z 535.448,A -85,B 0,C 180,E1 -15292.427,E2 -15292.427} C_VEL
LIN {X 0,Y 319.746,Z 535.47,A -85,B 0,C 180,E1 -15294.956,E2 -15294.956} C_VEL
LIN {X 0,Y 319.774,Z 535.74,A -85,B 0,C 180,E1 -15296.102,E2 -15296.102} C_VEL
LIN {X 0,Y 320.004,Z 536.638,A -85,B 0,C 180,E1 -15296.294,E2 -15296.294} C_VEL
LIN {X 0,Y 321.586,Z 539.355,A -85,B 0,C 180,E1 -15296.6,E2 -15296.6} C_VEL
LIN {X 0,Y 325.829,Z 546.833,A -85,B 0,C 180,E1 -15297.328,E2 -15297.328} C_VEL
LIN {X 0,Y 329.923,Z 554.991,A -85,B 0,C 180,E1 -15298.016,E2 -15298.016} C_VEL
LIN {X 0,Y 332.051,Z 560.303,A -85,B 0,C 180,E1 -15298.392,E2 -15298.392} C_VEL
LIN {X 0,Y 332.004,Z 579.497,A -85,B 0,C 180,E1 -15298.992,E2 -15298.992} C_VEL
LIN {X 0,Y 331.8,Z 591.065,A -85,B 0,C 180,E1 -15299.573,E2 -15299.573} C_VEL
LIN {X 0,Y 331.184,Z 603.114,A -85,B 0,C 180,E1 -15300.418,E2 -15300.418} C_VEL
LIN {X 0,Y 330.199,Z 614.494,A -85,B 0,C 180,E1 -15301.467,E2 -15301.467} C_VEL
LIN {X 0,Y 329.063,Z 625.224,A -85,B 0,C 180,E1 -15302.755,E2 -15302.755} C_VEL
LIN {X 0,Y 327.716,Z 635.42,A -85,B 0,C 180,E1 -15304.305,E2 -15304.305} C_VEL
LIN {X 0,Y 326.392,Z 643.629,A -85,B 0,C 180,E1 -15305.871,E2 -15305.871} C_VEL
LIN {X 0,Y 324.983,Z 651.508,A -85,B 0,C 180,E1 -15307.768,E2 -15307.768} C_VEL
LIN {X 0,Y 323.915,Z 656.82,A -85,B 0,C 180,E1 -15309.366,E2 -15309.366} C_VEL
LIN {X 0,Y 322.703,Z 662.269,A -85,B 0,C 180,E1 -15311.476,E2 -15311.476} C_VEL
LIN {X 0,Y 321.85,Z 665.663,A -85,B 0,C 180,E1 -15313.255,E2 -15313.255} C_VEL
LIN {X 0,Y 320.959,Z 668.591,A -85,B 0,C 180,E1 -15315.541,E2 -15315.541} C_VEL
LIN {X 0,Y 320.339,Z 670.069,A -85,B 0,C 180,E1 -15317.888,E2 -15317.888} C_VEL
LIN {X 0,Y 320.083,Z 670.231,A -85,B 0,C 180,E1 -15319.245,E2 -15319.245} C_VEL
LIN {X 0,Y 319.917,Z 669.941,A -85,B 0,C 180,E1 -15320.579,E2 -15320.579} C_VEL
LIN {X 0,Y 319.79,Z 668.528,A -85,B 0,C 180,E1 -15322.63,E2 -15322.63} C_VEL
LIN {X 0,Y 319.884,Z 665.979,A -85,B 0,C 180,E1 -15324.674,E2 -15324.674} C_VEL
LIN {X 0,Y 320.168,Z 662.176,A -85,B 0,C 180,E1 -15326.744,E2 -15326.744} C_VEL
LIN {X 0,Y 320.536,Z 656.963,A -85,B 0,C 180,E1 -15328.841,E2 -15328.841} C_VEL
LIN {X 0,Y 321.127,Z 650.032,A -85,B 0,C 180,E1 -15330.952,E2 -15330.952} C_VEL
LIN {X 0,Y 321.747,Z 642.724,A -85,B 0,C 180,E1 -15332.727,E2 -15332.727} C_VEL
LIN {X 0,Y 322.56,Z 633.562,A -85,B 0,C 180,E1 -15334.507,E2 -15334.507} C_VEL
LIN {X 0,Y 323.267,Z 624.459,A -85,B 0,C 180,E1 -15335.945,E2 -15335.945} C_VEL
LIN {X 0,Y 323.933,Z 614.155,A -85,B 0,C 180,E1 -15337.274,E2 -15337.274} C_VEL
LIN {X 0,Y 324.672,Z 602.133,A -85,B 0,C 180,E1 -15338.488,E2 -15338.488} C_VEL
LIN {X 0,Y 325.21,Z 590.357,A -85,B 0,C 180,E1 -15339.407,E2 -15339.407} C_VEL
LIN {X 0,Y 325.509,Z 577.365,A -85,B 0,C 180,E1 -15340.141,E2 -15340.141} C_VEL
LIN {X 0,Y 325.583,Z 563.997,A -85,B 0,C 180,E1 -15340.633,E2 -15340.633} C_VEL
LIN {X 0,Y 325.484,Z 553.864,A -85,B 0,C 180,E1 -15340.912,E2 -15340.912} C_VEL
LIN {X 0,Y 319.798,Z 536.578,A -85,B 0,C 180,E1 -15341.654,E2 -15341.654} C_VEL
LIN {X 0,Y 319.588,Z 535.591,A -85,B 0,C 180,E1 -15341.894,E2 -15341.894} C_VEL
LIN {X 0,Y 319.576,Z 535.492,A -85,B 0,C 180,E1 -15345.274,E2 -15345.274} C_VEL
LIN {X 0,Y 319.578,Z 535.487,A -85,B 0,C 180,E1 -15348.721,E2 -15348.721} C_VEL
LIN {X 0,Y 319.598,Z 535.484,A -85,B 0,C 180,E1 -15352.34,E2 -15352.34} C_VEL
LIN {X 0,Y 319.561,Z 535.491,A -85,B 0,C 180,E1 -15355.125,E2 -15355.125} C_VEL
LIN {X 0,Y 319.571,Z 535.489,A -85,B 0,C 180,E1 -15359.059,E2 -15359.059} C_VEL
LIN {X 0,Y 319.61,Z 535.482,A -85,B 0,C 180,E1 -15362.499,E2 -15362.499} C_VEL
LIN {X 0,Y 319.607,Z 535.486,A -85,B 0,C 180,E1 -15365.305,E2 -15365.305} C_VEL
LIN {X 0,Y 319.599,Z 535.485,A -85,B 0,C 180,E1 -15368.049,E2 -15368.049} C_VEL
LIN {X 0,Y 319.627,Z 535.482,A -85,B 0,C 180,E1 -15372.072,E2 -15372.072} C_VEL
LIN {X 0,Y 319.736,Z 535.469,A -85,B 0,C 180,E1 -15376.008,E2 -15376.008} C_VEL
LIN {X 0,Y 319.756,Z 535.468,A -85,B 0,C 180,E1 -15379.873,E2 -15379.873} C_VEL
LIN {X 0,Y 319.913,Z 535.45,A -85,B 0,C 180,E1 -15383.694,E2 -15383.694} C_VEL
LIN {X 0,Y 319.993,Z 535.438,A -85,B 0,C 180,E1 -15387.483,E2 -15387.483} C_VEL
LIN {X 0,Y 320.154,Z 535.418,A -85,B 0,C 180,E1 -15390,E2 -15390} C_VEL
LIN {X 0,Y 319.994,Z 535.435,A -85,B 0,C 180,E1 -15392.518,E2 -15392.518} C_VEL
LIN {X 0,Y 319.913,Z 535.446,A -85,B 0,C 180,E1 -15396.306,E2 -15396.306} C_VEL
LIN {X 0,Y 319.74,Z 535.469,A -85,B 0,C 180,E1 -15400.128,E2 -15400.128} C_VEL
LIN {X 0,Y 319.736,Z 535.471,A -85,B 0,C 180,E1 -15403.992,E2 -15403.992} C_VEL
LIN {X 0,Y 319.662,Z 535.481,A -85,B 0,C 180,E1 -15407.926,E2 -15407.926} C_VEL
LIN {X 0,Y 319.607,Z 535.483,A -85,B 0,C 180,E1 -15410.599,E2 -15410.599} C_VEL
LIN {X 0,Y 319.605,Z 535.483,A -85,B 0,C 180,E1 -15414.695,E2 -15414.695} C_VEL
LIN {X 0,Y 319.613,Z 535.484,A -85,B 0,C 180,E1 -15418.409,E2 -15418.409} C_VEL
LIN {X 0,Y 319.533,Z 535.496,A -85,B 0,C 180,E1 -15421.861,E2 -15421.861} C_VEL
LIN {X 0,Y 319.581,Z 535.487,A -85,B 0,C 180,E1 -15425.542,E2 -15425.542} C_VEL
LIN {X 0,Y 319.6,Z 535.489,A -85,B 0,C 180,E1 -15428.003,E2 -15428.003} C_VEL
LIN {X 0,Y 319.597,Z 535.485,A -85,B 0,C 180,E1 -15431.611,E2 -15431.611} C_VEL
LIN {X 0,Y 319.544,Z 535.49,A -85,B 0,C 180,E1 -15435.266,E2 -15435.266} C_VEL
LIN {X 0,Y 319.527,Z 535.494,A -85,B 0,C 180,E1 -15438.711,E2 -15438.711} C_VEL
LIN {X 0,Y 319.575,Z 535.491,A -85,B 0,C 180,E1 -15442.343,E2 -15442.343} C_VEL
LIN {X 0,Y 319.557,Z 535.488,A -85,B 0,C 180,E1 -15445.122,E2 -15445.122} C_VEL
LIN {X 0,Y 319.572,Z 535.487,A -85,B 0,C 180,E1 -15449.056,E2 -15449.056} C_VEL
LIN {X 0,Y 319.6,Z 535.485,A -85,B 0,C 180,E1 -15452.289,E2 -15452.289} C_VEL
LIN {X 0,Y 318.959,Z 535.57,A -85,B 0,C 180,E1 -15453.34,E2 -15453.34} C_VEL
LIN {X 0,Y 316.139,Z 535.923,A -85,B 0,C 180,E1 -15455.052,E2 -15455.052} C_VEL
LIN {X 0,Y 313.72,Z 536.22,A -85,B 0,C 180,E1 -15456.439,E2 -15456.439} C_VEL
LIN {X 0,Y 312.658,Z 536.348,A -85,B 0,C 180,E1 -15457.513,E2 -15457.513} C_VEL
LIN {X 0,Y 312.559,Z 536.359,A -85,B 0,C 180,E1 -15457.877,E2 -15457.877} C_VEL
LIN {X 0,Y 312.634,Z 536.352,A -85,B 0,C 180,E1 -15461.656,E2 -15461.656} C_VEL
LIN {X 0,Y 312.689,Z 536.345,A -85,B 0,C 180,E1 -15465.685,E2 -15465.685} C_VEL
LIN {X 0,Y 312.698,Z 536.343,A -85,B 0,C 180,E1 -15469.641,E2 -15469.641} C_VEL
LIN {X 0,Y 312.866,Z 536.326,A -85,B 0,C 180,E1 -15472.254,E2 -15472.254} C_VEL
LIN {X 0,Y 312.713,Z 536.343,A -85,B 0,C 180,E1 -15474.842,E2 -15474.842} C_VEL
LIN {X 0,Y 312.984,Z 536.311,A -85,B 0,C 180,E1 -15478.713,E2 -15478.713} C_VEL
LIN {X 0,Y 312.984,Z 536.308,A -85,B 0,C 180,E1 -15481.286,E2 -15481.286} C_VEL
LIN {X 0,Y 312.71,Z 536.342,A -85,B 0,C 180,E1 -15485.157,E2 -15485.157} C_VEL
LIN {X 0,Y 312.859,Z 536.323,A -85,B 0,C 180,E1 -15487.746,E2 -15487.746} C_VEL
LIN {X 0,Y 312.662,Z 536.348,A -85,B 0,C 180,E1 -15491.671,E2 -15491.671} C_VEL
LIN {X 0,Y 312.693,Z 536.347,A -85,B 0,C 180,E1 -15494.887,E2 -15494.887} C_VEL
LIN {X 0,Y 312.603,Z 536.356,A -85,B 0,C 180,E1 -15499.225,E2 -15499.225} C_VEL
LIN {X 0,Y 312.52,Z 536.37,A -85,B 0,C 180,E1 -15502.78,E2 -15502.78} C_VEL
LIN {X 0,Y 312.577,Z 536.364,A -85,B 0,C 180,E1 -15506.723,E2 -15506.723} C_VEL
LIN {X 0,Y 312.539,Z 536.363,A -85,B 0,C 180,E1 -15509.65,E2 -15509.65} C_VEL
LIN {X 0,Y 312.514,Z 536.366,A -85,B 0,C 180,E1 -15513.689,E2 -15513.689} C_VEL
LIN {X 0,Y 312.515,Z 536.367,A -85,B 0,C 180,E1 -15517.386,E2 -15517.386} C_VEL
LIN {X 0,Y 312.485,Z 536.374,A -85,B 0,C 180,E1 -15520.709,E2 -15520.709} C_VEL
LIN {X 0,Y 312.468,Z 536.372,A -85,B 0,C 180,E1 -15524.206,E2 -15524.206} C_VEL
LIN {X 0,Y 312.482,Z 536.37,A -85,B 0,C 180,E1 -15527.919,E2 -15527.919} C_VEL
LIN {X 0,Y 312.502,Z 536.368,A -85,B 0,C 180,E1 -15531.918,E2 -15531.918} C_VEL
LIN {X 0,Y 312.639,Z 536.479,A -85,B 0,C 180,E1 -15534.433,E2 -15534.433} C_VEL
LIN {X 0,Y 315.222,Z 549.844,A -85,B 0,C 180,E1 -15538.617,E2 -15538.617} C_VEL
LIN {X 0,Y 316.196,Z 555.897,A -85,B 0,C 180,E1 -15540.419,E2 -15540.419} C_VEL
LIN {X 0,Y 314.444,Z 570.42,A -85,B 0,C 180,E1 -15544.517,E2 -15544.517} C_VEL
LIN {X 0,Y 312.82,Z 587.391,A -85,B 0,C 180,E1 -15549.278,E2 -15549.278} C_VEL
LIN {X 0,Y 312.554,Z 590.843,A -85,B 0,C 180,E1 -15550.203,E2 -15550.203} C_VEL
LIN {X 0,Y 312.81,Z 595.54,A -85,B 0,C 180,E1 -15550.43,E2 -15550.43} C_VEL
LIN {X 0,Y 316.821,Z 650.777,A -85,B 0,C 180,E1 -15552.354,E2 -15552.354} C_VEL
LIN {X 0,Y 316.12,Z 676.61,A -85,B 0,C 180,E1 -15553.201,E2 -15553.201} C_VEL
LIN {X 0,Y 315.592,Z 688.55,A -85,B 0,C 180,E1 -15553.838,E2 -15553.838} C_VEL
LIN {X 0,Y 314.701,Z 699.067,A -85,B 0,C 180,E1 -15554.622,E2 -15554.622} C_VEL
LIN {X 0,Y 313.866,Z 708.857,A -85,B 0,C 180,E1 -15555.576,E2 -15555.576} C_VEL
LIN {X 0,Y 313.208,Z 717.979,A -85,B 0,C 180,E1 -15556.703,E2 -15556.703} C_VEL
LIN {X 0,Y 312.472,Z 726.431,A -85,B 0,C 180,E1 -15557.992,E2 -15557.992} C_VEL
LIN {X 0,Y 311.904,Z 734.905,A -85,B 0,C 180,E1 -15559.615,E2 -15559.615} C_VEL
LIN {X 0,Y 311.659,Z 741.711,A -85,B 0,C 180,E1 -15561.245,E2 -15561.245} C_VEL
LIN {X 0,Y 311.631,Z 747.127,A -85,B 0,C 180,E1 -15562.884,E2 -15562.884} C_VEL
LIN {X 0,Y 311.84,Z 752.05,A -85,B 0,C 180,E1 -15564.828,E2 -15564.828} C_VEL
LIN {X 0,Y 312.005,Z 754.5,A -85,B 0,C 180,E1 -15566.125,E2 -15566.125} C_VEL
LIN {X 0,Y 312.118,Z 756.341,A -85,B 0,C 180,E1 -15567.419,E2 -15567.419} C_VEL
LIN {X 0,Y 312.352,Z 757.573,A -85,B 0,C 180,E1 -15568.711,E2 -15568.711} C_VEL
LIN {X 0,Y 312.583,Z 758.276,A -85,B 0,C 180,E1 -15570,E2 -15570} C_VEL
LIN {X 0,Y 312.146,Z 758.29,A -85,B 0,C 180,E1 -15571.29,E2 -15571.29} C_VEL
LIN {X 0,Y 311.95,Z 757.826,A -85,B 0,C 180,E1 -15572.582,E2 -15572.582} C_VEL
LIN {X 0,Y 311.762,Z 756.798,A -85,B 0,C 180,E1 -15573.878,E2 -15573.878} C_VEL
LIN {X 0,Y 311.438,Z 754.258,A -85,B 0,C 180,E1 -15575.828,E2 -15575.828} C_VEL
LIN {X 0,Y 311.343,Z 750.438,A -85,B 0,C 180,E1 -15577.784,E2 -15577.784} C_VEL
LIN {X 0,Y 311.523,Z 745.267,A -85,B 0,C 180,E1 -15579.741,E2 -15579.741} C_VEL
LIN {X 0,Y 312.137,Z 738.595,A -85,B 0,C 180,E1 -15581.691,E2 -15581.691} C_VEL
LIN {X 0,Y 313.167,Z 731.659,A -85,B 0,C 180,E1 -15583.298,E2 -15583.298} C_VEL
LIN {X 0,Y 314.534,Z 723.141,A -85,B 0,C 180,E1 -15584.889,E2 -15584.889} C_VEL
LIN {X 0,Y 316.138,Z 712.495,A -85,B 0,C 180,E1 -15586.465,E2 -15586.465} C_VEL
LIN {X 0,Y 317.895,Z 701.692,A -85,B 0,C 180,E1 -15587.697,E2 -15587.697} C_VEL
LIN {X 0,Y 319.357,Z 690.812,A -85,B 0,C 180,E1 -15588.678,E2 -15588.678} C_VEL
LIN {X 0,Y 320.736,Z 678.38,A -85,B 0,C 180,E1 -15589.521,E2 -15589.521} C_VEL
LIN {X 0,Y 321.878,Z 664.519,A -85,B 0,C 180,E1 -15590.155,E2 -15590.155} C_VEL
LIN {X 0,Y 322.305,Z 649.549,A -85,B 0,C 180,E1 -15590.631,E2 -15590.631} C_VEL
LIN {X 0,Y 321.195,Z 623.51,A -85,B 0,C 180,E1 -15591.626,E2 -15591.626} C_VEL
LIN {X 0,Y 319.339,Z 606.238,A -85,B 0,C 180,E1 -15592.433,E2 -15592.433} C_VEL
LIN {X 0,Y 316.313,Z 587.218,A -85,B 0,C 180,E1 -15593.478,E2 -15593.478} C_VEL
LIN {X 0,Y 313.822,Z 574.719,A -85,B 0,C 180,E1 -15594.274,E2 -15594.274} C_VEL
LIN {X 0,Y 313.94,Z 572.498,A -85,B 0,C 180,E1 -15594.783,E2 -15594.783} C_VEL
LIN {X 0,Y 315.908,Z 556.973,A -85,B 0,C 180,E1 -15599.302,E2 -15599.302} C_VEL
LIN {X 0,Y 316.041,Z 553.985,A -85,B 0,C 180,E1 -15600.234,E2 -15600.234} C_VEL
LIN {X 0,Y 314.207,Z 544.081,A -85,B 0,C 180,E1 -15603.613,E2 -15603.613} C_VEL
LIN {X 0,Y 312.563,Z 536.454,A -85,B 0,C 180,E1 -15606.522,E2 -15606.522} C_VEL
LIN {X 0,Y 312.486,Z 536.372,A -85,B 0,C 180,E1 -15610.709,E2 -15610.709} C_VEL
LIN {X 0,Y 312.514,Z 536.367,A -85,B 0,C 180,E1 -15614.197,E2 -15614.197} C_VEL
LIN {X 0,Y 312.543,Z 536.358,A -85,B 0,C 180,E1 -15617.905,E2 -15617.905} C_VEL
LIN {X 0,Y 312.555,Z 536.362,A -85,B 0,C 180,E1 -15621.904,E2 -15621.904} C_VEL
LIN {X 0,Y 312.501,Z 536.371,A -85,B 0,C 180,E1 -15625.79,E2 -15625.79} C_VEL
LIN {X 0,Y 312.522,Z 536.369,A -85,B 0,C 180,E1 -15628.854,E2 -15628.854} C_VEL
LIN {X 0,Y 312.568,Z 536.363,A -85,B 0,C 180,E1 -15631.825,E2 -15631.825} C_VEL
LIN {X 0,Y 312.578,Z 536.359,A -85,B 0,C 180,E1 -15634.711,E2 -15634.711} C_VEL
LIN {X 0,Y 312.58,Z 536.359,A -85,B 0,C 180,E1 -15637.529,E2 -15637.529} C_VEL
